(*=======================================================*)
	216:	(* Servobandeinzug rückwärts fahren, damit die Ausschiebezylinder das Band sicher erwischen *)
		IF fb_state_entry.E THEN
			axis_bandeinzug_achse.st_ctrl.in.b_ausfaedeln_servo := TRUE;
		END_IF

		(*-----------------------Weiterschaltbedingungen----------------------------*)
		IF axis_bandeinzug_achse.st_ctrl.out.b_ausgefaedelt_servo AND NOT fb_state_entry.E THEN
			axis_bandeinzug_achse.st_ctrl.in.b_ausfaedeln_servo := FALSE;
			fb_state_entry.i16_next_step := 217;(*Neu*)
		END_IF

(*=======================================================*)
	217:	(* Fänger ins Band fahren, damit die Bremse gelöst werden kann *)
		IF fb_state_entry.E THEN
				zyl_bawe_faenger_li.st_ctrl.in.b_ausfahren := TRUE;
		END_IF

		(*-----------------------Weiterschaltbedingungen----------------------------*)
		IF 	zyl_bawe_faenger_li.st_ctrl.out.b_ausgefahren AND
			gb_ba_auto_kontroller
			THEN
				zyl_bawe_faenger_li.st_ctrl.in.b_ausfahren := FALSE;
				fb_state_entry.i16_next_step := 218;
		END_IF

(*=======================================================*)
	218:	(* Bremse an Servobandeinzug lösen, damit Band heraus gezogen werden kann. Die Bestückachse hat die Slavekopplung bereits gelöst. *)
		IF fb_state_entry.E THEN
			axis_bandeinzug_achse.st_ctrl.in.b_bremse_auf := TRUE;
		END_IF

		(*-----------------------Weiterschaltbedingungen----------------------------*)
		IF axis_bandeinzug_achse.st_ctrl.out.b_bremse_geoeffnet AND NOT fb_state_entry.E THEN
			axis_bandeinzug_achse.st_ctrl.in.b_bremse_auf := FALSE;
			fb_state_entry.i16_next_step := 220;
		END_IF

(*=======================================================*)
	220:	(* Vorschub einfahren und Band aus WKZ rausziehen *)
		IF fb_state_entry.E THEN
			zyl_bawe_vorschub.st_ctrl.in.b_einfahren := TRUE;
			i16_akt_ausfaedeln := i16_akt_ausfaedeln + 1;
		END_IF

		(*-----------------------Weiterschaltbedingungen----------------------------*)
		IF zyl_bawe_vorschub.st_ctrl.out.b_eingefahren AND gb_ba_auto_kontroller THEN
			zyl_bawe_vorschub.st_ctrl.in.b_einfahren := FALSE;
			IF i16_akt_ausfaedeln <= i16_vorgabe_ausfaedeln THEN
				fb_state_entry.i16_next_step := 230;
			ELSE
				fb_state_entry.i16_next_step := 280;
			END_IF
		END_IF

(*=======================================================*)
	230:	(* Bandwechselhalter links ausfahren um Band nachfassen zu können *)
		IF fb_state_entry.E THEN
			zyl_bawe_halter_li.st_ctrl.in.b_ausfahren := TRUE;
		END_IF

		(*-----------------------Weiterschaltbedingungen----------------------------*)
		IF zyl_bawe_halter_li.st_ctrl.out.b_ausgefahren AND gb_ba_auto_kontroller THEN
			zyl_bawe_halter_li.st_ctrl.in.b_ausfahren := FALSE;
			fb_state_entry.i16_next_step := 240;
		END_IF

(*=======================================================*)
	240:	(* Bandwechselfänger links einfahren*)
		IF fb_state_entry.E THEN
			zyl_bawe_faenger_li.st_ctrl.in.b_einfahren := TRUE;
		END_IF

		(*-----------------------Weiterschaltbedingungen----------------------------*)
		IF zyl_bawe_faenger_li.st_ctrl.out.b_eingefahren AND gb_ba_auto_kontroller THEN
			zyl_bawe_faenger_li.st_ctrl.in.b_einfahren := FALSE;
			fb_state_entry.i16_next_step := 250;
		END_IF

(*=======================================================*)
	250:	(* Vorschub ausfahren und Band nachfassen *)
		IF fb_state_entry.E THEN
			zyl_bawe_vorschub.st_ctrl.in.b_ausfahren := TRUE;
		END_IF

		(*-----------------------Weiterschaltbedingungen----------------------------*)
		IF zyl_bawe_vorschub.st_ctrl.out.b_ausgefahren AND gb_ba_auto_kontroller THEN
			zyl_bawe_vorschub.st_ctrl.in.b_ausfahren := FALSE;
			fb_state_entry.i16_next_step := 260;
		END_IF

(*=======================================================*)
	260:	(* Bandwechselfänger links ausfahren zum Band halten *)
		IF fb_state_entry.E THEN
			zyl_bawe_faenger_li.st_ctrl.in.b_ausfahren := TRUE;
		END_IF

		(*-----------------------Weiterschaltbedingungen----------------------------*)
		IF zyl_bawe_faenger_li.st_ctrl.out.b_ausgefahren AND gb_ba_auto_kontroller THEN
			zyl_bawe_faenger_li.st_ctrl.in.b_ausfahren := FALSE;
			fb_state_entry.i16_next_step := 270;
		END_IF

(*=======================================================*)
	270:	(* Bandwechselhalter links einfahren und Band freigeben*)
		IF fb_state_entry.E THEN
			zyl_bawe_halter_li.st_ctrl.in.b_einfahren := TRUE;
		END_IF

		(*-----------------------Weiterschaltbedingungen----------------------------*)
		IF zyl_bawe_halter_li.st_ctrl.out.b_eingefahren AND gb_ba_auto_kontroller THEN
			zyl_bawe_halter_li.st_ctrl.in.b_einfahren := FALSE;
			fb_state_entry.i16_next_step := 220;
		END_IF

(*=======================================================*)
	280:	(* Fänger links einfahren zum Ausfädeln *)
		IF fb_state_entry.E THEN
			zyl_bawe_faenger_li.st_ctrl.in.b_einfahren := TRUE;
		END_IF

		(*-----------------------Weiterschaltbedingungen----------------------------*)
		IF zyl_bawe_faenger_li.st_ctrl.out.b_eingefahren AND gb_ba_auto_kontroller THEN
			zyl_bawe_faenger_li.st_ctrl.in.b_einfahren := FALSE;
			fb_state_entry.i16_next_step := 290;
		END_IF

(*=======================================================*)
	290:	(* Band ist herausgezogen - prüfe Einstellung bzw. Bandanwesenheit im rechten Einzug *)
		b_ausgefaedelt:=b_materialmangel;
			(* Band vorhanden -> Beginn automatischer Bandwechsel *)
		(*-----------------------Weiterschaltbedingungen----------------------------*)
		IF fb_tof_bandende_re.Q AND gst_datensatz.st_md.b_auto_Bandwechsel THEN
			b_spulenwechsel := TRUE;
			fb_state_entry.i16_next_step := 300;
		ELSE
			(* Bandherausziehen ist fertig *)
			fb_state_entry.i16_next_step := 295;
		END_IF

(*=======================================================*)
	291:	(* Bediener muss am Backpanel auswählen ob Bandwechsel oder Trennstelle *)

		(*-----------------------Weiterschaltbedingungen----------------------------*)
		IF visu_hinten.out.b_Bandwechsel THEN
			(* Band vorhanden -> Beginn automatischer Bandwechsel *)
			visu_hinten.in.b_bandwechsel_aktiv := FALSE;
			visu_hinten.in.current_visu_folie := 'BESTUECKZELLE_1700';
			fb_state_entry.i16_next_step := 300;
		ELSIF visu_hinten.out.b_Trennstelle THEN
			visu_hinten.in.b_bandwechsel_aktiv := FALSE;
			CASE gst_datensatz.st_wkz.i16_typ_bandeinzug OF

				 BANDWECHSLER_V2:
					visu_hinten.in.current_visu_folie := 'BA_1700_BAND_EINFAEDELN';

				SERVO:
					visu_hinten.in.current_visu_folie := 'BA1700_SERVO_BAND_EINFAEDELN';
			END_CASE
			fb_state_entry.i16_next_step := 295;
		END_IF

(*=======================================================*)
	295:	(* Vorschub ausfahren und fertig -> Band wird jetzt im gleichen Einzug manuell eingelegt mit Einfädelprozedur in der Bestückachse *)
		IF fb_state_entry.E THEN
			zyl_bawe_vorschub.st_ctrl.in.b_ausfahren := TRUE;
		END_IF

		(*-----------------------Weiterschaltbedingungen----------------------------*)
		IF zyl_bawe_vorschub.st_ctrl.out.b_ausgefahren AND gb_ba_auto_kontroller THEN
			zyl_bawe_vorschub.st_ctrl.in.b_ausfahren := FALSE;
			st_ctrl_out.b_fertig_2 := TRUE;
			fb_state_entry.i16_next_step := BEREIT;
		END_IF

(*=======================================================*)
	300:	(* Fänger rechts ausfahren *)
		IF fb_state_entry.E THEN
			zyl_bawe_faenger_re.st_ctrl.in.b_ausfahren := TRUE;
		END_IF

		(*-----------------------Weiterschaltbedingungen----------------------------*)
		IF 	zyl_bawe_faenger_re.st_ctrl.out.b_ausgefahren AND
			gb_ba_auto_kontroller
			THEN
				zyl_bawe_faenger_re.st_ctrl.in.b_ausfahren := FALSE;
				fb_state_entry.i16_next_step := 310;
		END_IF

(*=======================================================*)
	310:	(* Halter rechts einfahren *)
		IF fb_state_entry.E THEN
			zyl_bawe_halter_re.st_ctrl.in.b_einfahren := TRUE;
		END_IF

		(*-----------------------Weiterschaltbedingungen----------------------------*)
		IF zyl_bawe_halter_re.st_ctrl.out.b_eingefahren AND gb_ba_auto_kontroller THEN
			zyl_bawe_halter_re.st_ctrl.in.b_einfahren := FALSE;
			fb_state_entry.i16_next_step := 315;
		END_IF

(*=======================================================*)
	315:	(* Spulenbremse rechts oben? *)

		(*-----------------------Weiterschaltbedingungen----------------------------*)
		IF zyl_haspel_re_abspulen.st_ctrl.out.b_ausgefahren AND gb_ba_auto_kontroller THEN
			fb_state_entry.i16_next_step := 320;
		END_IF

(*=======================================================*)
	320:	(* Querschub ausfahren -> nach links und Haspeln nach links: Haspel verschieben ausfahren und Bandabzug einfahren *)
		IF fb_state_entry.E THEN
			zyl_bawe_querschub.st_ctrl.in.b_ausfahren := TRUE;
			zyl_haspel_verschieben.st_ctrl.in.b_ausfahren := TRUE;
			zyl_bandeinzuege_verschieben.st_ctrl.in.b_einfahren := TRUE;
		END_IF

		(*-----------------------Weiterschaltbedingungen----------------------------*)
		IF 	zyl_bawe_querschub.st_ctrl.out.b_ausgefahren AND
			zyl_haspel_verschieben.st_ctrl.out.b_ausgefahren AND
			zyl_bandeinzuege_verschieben.st_ctrl.out.b_eingefahren AND
			gb_ba_auto_kontroller
			THEN
				zyl_bawe_querschub.st_ctrl.in.b_ausfahren := FALSE;
				zyl_haspel_verschieben.st_ctrl.in.b_ausfahren := FALSE;
				zyl_bandeinzuege_verschieben.st_ctrl.in.b_einfahren := FALSE;
				CASE gst_datensatz.st_wkz.i16_typ_bandeinzug OF

					BANDWECHSLER_V2:
						fb_state_entry.i16_next_step := 330;

					SERVO:
						fb_state_entry.i16_next_step := 325;
				END_CASE
		END_IF

		IF fb_state_entry.X THEN
			b_spulenwechsel := FALSE;
		END_IF

(*=======================================================*)
	325:	(* Igelrad auf Position *)
		IF fb_state_entry.E THEN
			axis_bandeinzug_achse.st_ctrl.in.b_startpos := TRUE;
			fb_ton_wz.PT := t#100ms;
			fb_ton_wz.IN := TRUE;
		END_IF

		(*-----------------------Weiterschaltbedingungen----------------------------*)
		IF axis_bandeinzug_achse.st_ctrl.out.b_servo_auf_einfaedelpos
		AND gb_ba_auto_kontroller AND fb_ton_wz.Q THEN
			axis_bandeinzug_achse.st_ctrl.in.b_startpos := FALSE;
			fb_state_entry.i16_next_step := 330;
		END_IF

		IF fb_state_entry.X THEN
			fb_ton_wz.IN := FALSE;
		END_IF

(*=======================================================*)
	330:	(* Vorschub ausfahren *)
		IF fb_state_entry.E THEN
			zyl_bawe_vorschub.st_ctrl.in.b_ausfahren := TRUE;
			i16_akt_einfaedeln := i16_akt_einfaedeln + 1;
		END_IF

		(*-----------------------Weiterschaltbedingungen----------------------------*)
		IF zyl_bawe_vorschub.st_ctrl.out.b_ausgefahren AND gb_ba_auto_kontroller THEN
			zyl_bawe_vorschub.st_ctrl.in.b_ausfahren := FALSE;
			IF i16_akt_einfaedeln < i16_vorgabe_einfaedeln THEN
				fb_state_entry.i16_next_step := 340;
			ELSE
				fb_state_entry.i16_next_step := 390;		 (*mit Wartezeit alt 400*)
			END_IF
		END_IF

(*=======================================================*)
	340:	(* Halter rechts ausfahren *)
		IF fb_state_entry.E THEN
			zyl_bawe_halter_re.st_ctrl.in.b_ausfahren := TRUE;
		END_IF

		(*-----------------------Weiterschaltbedingungen----------------------------*)
		IF zyl_bawe_halter_re.st_ctrl.out.b_ausgefahren AND gb_ba_auto_kontroller THEN
			zyl_bawe_halter_re.st_ctrl.in.b_ausfahren := FALSE;
			fb_state_entry.i16_next_step := 350;
		END_IF

(*=======================================================*)
	350:	(* Fänger rechts einfahren *)
		IF fb_state_entry.E THEN
			zyl_bawe_faenger_re.st_ctrl.in.b_einfahren := TRUE;
		END_IF

		(*-----------------------Weiterschaltbedingungen----------------------------*)
		IF zyl_bawe_faenger_re.st_ctrl.out.b_eingefahren AND gb_ba_auto_kontroller THEN
			zyl_bawe_faenger_re.st_ctrl.in.b_einfahren := FALSE;
			fb_state_entry.i16_next_step := 360;
		END_IF

(*=======================================================*)
	360:	(* Vorschub einfahren *)
		IF fb_state_entry.E THEN
			zyl_bawe_vorschub.st_ctrl.in.b_einfahren := TRUE;
		END_IF

		(*-----------------------Weiterschaltbedingungen----------------------------*)
		IF zyl_bawe_vorschub.st_ctrl.out.b_eingefahren AND gb_ba_auto_kontroller THEN
			zyl_bawe_vorschub.st_ctrl.in.b_einfahren := FALSE;
			fb_state_entry.i16_next_step := 370;
		END_IF

(*=======================================================*)
	370:	(* Fänger rechts ausfahren *)
		IF fb_state_entry.E THEN
			zyl_bawe_faenger_re.st_ctrl.in.b_ausfahren := TRUE;
		END_IF

		(*-----------------------Weiterschaltbedingungen----------------------------*)
		IF zyl_bawe_faenger_re.st_ctrl.out.b_ausgefahren AND gb_ba_auto_kontroller THEN
			zyl_bawe_faenger_re.st_ctrl.in.b_ausfahren := FALSE;
			fb_state_entry.i16_next_step := 380;
		END_IF

(*=======================================================*)
	380:	(* Halter rechts einfahren *)
		IF fb_state_entry.E THEN
			zyl_bawe_halter_re.st_ctrl.in.b_einfahren := TRUE;
		END_IF

		(*-----------------------Weiterschaltbedingungen----------------------------*)
		IF zyl_bawe_halter_re.st_ctrl.out.b_eingefahren AND gb_ba_auto_kontroller THEN
			zyl_bawe_halter_re.st_ctrl.in.b_einfahren := FALSE;
			fb_state_entry.i16_next_step := 330;
		END_IF

(*=======================================================*)
	390:	(* Wartezeit damit der Fänger vom WZ trifft*)
		IF	 fb_state_entry.E THEN
			fb_ton_wz.IN:=FALSE;
		END_IF
		fb_ton_wz(IN:=TRUE,PT:=t#1000ms);
		(*-----------------------Weiterschaltbedingungen----------------------------*)
		IF 	fb_ton_wz.Q THEN
			fb_ton_wz.IN:=FALSE;
			fb_state_entry.i16_next_step := 400;
		END_IF

(*=======================================================*)
	400:	(* Nocken für Zylinder am Bandeinzug einschalten und somit Bandfänger ausfahren bzw. Bremse an Servobandeinzug wieder fest machen. *)

		CASE gst_datensatz.st_wkz.i16_typ_bandeinzug OF

			BANDWECHSLER_V2:

				IF fb_state_entry.E THEN
					(* Bandwechsler V2 ohne Sensoren und anderen Zylindern *)
					gst_datensatz.st_wkz.nockenschaltwerk_bestueckachse.arr_nocken[NO_BW_BANDFAENGER_BAWEV2_EINFAHREN].b_camvalid := TRUE;
					gst_datensatz.st_wkz.nockenschaltwerk_bestueckachse.arr_nocken[NO_BW_BANDFAENGER_BAWEV2_AUSFAHREN].b_camvalid := TRUE;
					gst_datensatz.st_wkz.nockenschaltwerk_bestueckachse.arr_nocken[NO_BW_BANDKLEMMEN_BAWEV2_EINFAHREN].b_camvalid := TRUE;
					gst_datensatz.st_wkz.nockenschaltwerk_bestueckachse.arr_nocken[NO_BW_BANDKLEMMEN_BAWEV2_AUSFAHREN].b_camvalid := TRUE;

					gst_datensatz.st_wkz.nockenschaltwerk_bestueckachse.arr_nocken[NO_PNEUMATIKBANDEINZUG_GLS].b_camvalid := TRUE;

					zyl_bandfaenger.fb.b_no_gesteuert_im_norm_betrieb := FALSE;
					zyl_bandklemmen.fb.b_no_gesteuert_im_norm_betrieb := FALSE;
					fb_ton_wz.PT := t#500ms;
					fb_ton_wz.IN := TRUE;
				END_IF

				(*-----------------------Weiterschaltbedingungen----------------------------*)
				IF fb_ton_wz.Q THEN
					fb_ton_wz.IN := FALSE;
					fb_state_entry.i16_next_step := 410;
				END_IF

			SERVO:
				IF fb_state_entry.E THEN
					axis_bandeinzug_achse.st_ctrl.in.b_bremse_auf := TRUE;	(* Bremse auf zum Position übernehmen *)
				END_IF

				(*-----------------------Weiterschaltbedingungen----------------------------*)
				IF axis_bandeinzug_achse.st_ctrl.out.b_bremse_geoeffnet THEN
					axis_bandeinzug_achse.st_ctrl.in.b_bremse_auf := FALSE;
					fb_state_entry.i16_next_step := 410;
				END_IF
		END_CASE;

(*=======================================================*)
	410:	(* Fänger rechts einfahren *)
		IF fb_state_entry.E THEN
			zyl_bawe_faenger_re.st_ctrl.in.b_einfahren := TRUE;
		END_IF

		(*-----------------------Weiterschaltbedingungen----------------------------*)
		IF zyl_bawe_faenger_re.st_ctrl.out.b_eingefahren
		AND gb_ba_auto_kontroller THEN
			zyl_bawe_faenger_re.st_ctrl.in.b_einfahren := FALSE;
			(* Bandwechsel ist fertig *)
			st_ctrl_out.b_fertig := TRUE;
			fb_state_entry.i16_next_step := BEREIT;
		END_IF


(*---------------------------------------------------------------------------------------------------------------------------------------------------------------------------------------------------*)
(*========================Bandeinzug rechts ist leer===============================*)
	500:	(* Fänger links ausfahren zum Band halten, Fänger rechts einfahren zur Bandfreigabe im rechten Einzug - Halter gegensinnig *)
		IF fb_state_entry.E THEN
			zyl_bawe_faenger_re.st_ctrl.in.b_ausfahren := TRUE;
			zyl_bawe_faenger_li.st_ctrl.in.b_einfahren := TRUE;
			zyl_bawe_halter_re.st_ctrl.in.b_einfahren := TRUE;
			zyl_bawe_halter_li.st_ctrl.in.b_ausfahren := TRUE;
		END_IF

		(*-----------------------Weiterschaltbedingungen----------------------------*)
		IF 	zyl_bawe_faenger_re.st_ctrl.out.b_ausgefahren AND
			zyl_bawe_faenger_li.st_ctrl.out.b_eingefahren AND
			zyl_bawe_halter_re.st_ctrl.out.b_eingefahren AND
			zyl_bawe_halter_li.st_ctrl.out.b_ausgefahren AND
			gb_ba_auto_kontroller
			THEN
				zyl_bawe_faenger_re.st_ctrl.in.b_ausfahren := FALSE;
				zyl_bawe_faenger_li.st_ctrl.in.b_einfahren := FALSE;
				zyl_bawe_halter_re.st_ctrl.in.b_einfahren := FALSE;
				zyl_bawe_halter_li.st_ctrl.in.b_ausfahren := FALSE;
				fb_state_entry.i16_next_step := 510;
		END_IF

(*=======================================================*)
	510:	(* Band-Zylinder einfahren bzw. Servobandeinzug lösen *)
		CASE gst_datensatz.st_wkz.i16_typ_bandeinzug OF
			BANDWECHSLER_V2:
				IF fb_state_entry.E THEN
					(* Zylinder einfahren *)
					zyl_bandfaenger.st_ctrl.in.b_einfahren := TRUE;
					zyl_bandklemmen.st_ctrl.in.b_einfahren := TRUE;
				END_IF

				(*-----------------------Weiterschaltbedingungen----------------------------*)
				IF 	zyl_bandfaenger.st_ctrl.out.b_eingefahren AND
					zyl_bandklemmen.st_ctrl.out.b_eingefahren AND
					gb_ba_auto_kontroller
					THEN
						zyl_bandfaenger.st_ctrl.in.b_einfahren := FALSE;
						zyl_bandklemmen.st_ctrl.in.b_einfahren := FALSE;
						fb_state_entry.i16_next_step := 520;
				END_IF

			SERVO:
				zyl_bawe_faenger_re.st_ctrl.in.b_einfahren := TRUE;
				zyl_bawe_halter_re.st_ctrl.in.b_einfahren := TRUE;
				(*-----------------------Weiterschaltbedingungen----------------------------*)
				IF 	zyl_bawe_faenger_re.st_ctrl.out.b_eingefahren AND
					zyl_bawe_halter_re.st_ctrl.out.b_eingefahren AND
					gb_ba_auto_kontroller
					THEN
						zyl_bawe_faenger_re.st_ctrl.in.b_einfahren := FALSE;
						zyl_bawe_halter_re.st_ctrl.in.b_einfahren := FALSE;
						fb_state_entry.i16_next_step := 516;
				END_IF
		END_CASE;

(*=======================================================*)
	516:	(* Servobandeinzug rückwärts fahren, damit die Ausschiebezylinder das Band sicher erwischen *)
		IF fb_state_entry.E THEN
			axis_bandeinzug_achse.st_ctrl.in.b_ausfaedeln_servo := TRUE;
		END_IF

		(*-----------------------Weiterschaltbedingungen----------------------------*)
		IF axis_bandeinzug_achse.st_ctrl.out.b_ausgefaedelt_servo AND NOT fb_state_entry.E THEN
			axis_bandeinzug_achse.st_ctrl.in.b_ausfaedeln_servo := FALSE;
			fb_state_entry.i16_next_step := 517;(*Neu*)
		END_IF

(*=======================================================*)
	517:	(* Fänger ins Band fahren, damit die Bremse gelöst werden kann *)
		IF fb_state_entry.E THEN
				zyl_bawe_faenger_re.st_ctrl.in.b_ausfahren := TRUE;
		END_IF

		(*-----------------------Weiterschaltbedingungen----------------------------*)
		IF 	zyl_bawe_faenger_re.st_ctrl.out.b_ausgefahren AND
			gb_ba_auto_kontroller
			THEN
				zyl_bawe_faenger_re.st_ctrl.in.b_ausfahren := FALSE;
				fb_state_entry.i16_next_step := 518;
		END_IF

(*=======================================================*)
	518:	(* Bremse an Servobandeinzug lösen, damit Band heraus gezogen werden kann. Die Bestückachse hat die Slavekopplung bereits gelöst. *)
		IF fb_state_entry.E THEN
			axis_bandeinzug_achse.st_ctrl.in.b_bremse_auf := TRUE;
		END_IF

		(*-----------------------Weiterschaltbedingungen----------------------------*)
		IF axis_bandeinzug_achse.st_ctrl.out.b_bremse_geoeffnet AND NOT fb_state_entry.E THEN
			axis_bandeinzug_achse.st_ctrl.in.b_bremse_auf := FALSE;
			fb_state_entry.i16_next_step := 520;
		END_IF

(*=======================================================*)
	520:	(* Vorschub einfahren und Band aus WKZ rausziehen *)
		IF fb_state_entry.E THEN
			zyl_bawe_vorschub.st_ctrl.in.b_einfahren := TRUE;
			i16_akt_ausfaedeln := i16_akt_ausfaedeln + 1;
		END_IF

		(*-----------------------Weiterschaltbedingungen----------------------------*)
		IF zyl_bawe_vorschub.st_ctrl.out.b_eingefahren AND gb_ba_auto_kontroller THEN
			zyl_bawe_vorschub.st_ctrl.in.b_einfahren := FALSE;
			IF i16_akt_ausfaedeln <= i16_vorgabe_ausfaedeln THEN
				fb_state_entry.i16_next_step := 530;
			ELSE
				fb_state_entry.i16_next_step := 580;
			END_IF
		END_IF

(*=======================================================*)
	530:	(* Bandwechselhalter rechts ausfahren um Band nachfassen zu können *)
		IF fb_state_entry.E THEN
			zyl_bawe_halter_re.st_ctrl.in.b_ausfahren := TRUE;
		END_IF

		(*-----------------------Weiterschaltbedingungen----------------------------*)
		IF zyl_bawe_halter_re.st_ctrl.out.b_ausgefahren AND gb_ba_auto_kontroller THEN
			zyl_bawe_halter_re.st_ctrl.in.b_ausfahren := FALSE;
			fb_state_entry.i16_next_step := 540;
		END_IF

(*=======================================================*)
	540:	(* Bandwechselfänger rechts einfahren*)
		IF fb_state_entry.E THEN
			zyl_bawe_faenger_re.st_ctrl.in.b_einfahren := TRUE;
		END_IF

		(*-----------------------Weiterschaltbedingungen----------------------------*)
		IF zyl_bawe_faenger_re.st_ctrl.out.b_eingefahren AND gb_ba_auto_kontroller THEN
			zyl_bawe_faenger_re.st_ctrl.in.b_einfahren := FALSE;
			fb_state_entry.i16_next_step := 550;
		END_IF

(*=======================================================*)
	550:	(* Vorschub ausfahren und Band nachfassen *)
		IF fb_state_entry.E THEN
			zyl_bawe_vorschub.st_ctrl.in.b_ausfahren := TRUE;
		END_IF

		(*-----------------------Weiterschaltbedingungen----------------------------*)
		IF zyl_bawe_vorschub.st_ctrl.out.b_ausgefahren AND gb_ba_auto_kontroller THEN
			zyl_bawe_vorschub.st_ctrl.in.b_ausfahren := FALSE;
			fb_state_entry.i16_next_step := 560;
		END_IF

(*=======================================================*)
	560:	(* Bandwechselfänger rechts ausfahren zum Band halten *)
		IF fb_state_entry.E THEN
			zyl_bawe_faenger_re.st_ctrl.in.b_ausfahren := TRUE;
		END_IF

		(*-----------------------Weiterschaltbedingungen----------------------------*)
		IF zyl_bawe_faenger_re.st_ctrl.out.b_ausgefahren AND gb_ba_auto_kontroller THEN
			zyl_bawe_faenger_re.st_ctrl.in.b_ausfahren := FALSE;
			fb_state_entry.i16_next_step := 570;
		END_IF

(*=======================================================*)
	570:	(* Bandwechselhalter rechts einfahren und Band freigeben*)
		IF fb_state_entry.E THEN
			zyl_bawe_halter_re.st_ctrl.in.b_einfahren := TRUE;
		END_IF

		(*-----------------------Weiterschaltbedingungen----------------------------*)
		IF zyl_bawe_halter_re.st_ctrl.out.b_eingefahren AND gb_ba_auto_kontroller THEN
			zyl_bawe_halter_re.st_ctrl.in.b_einfahren := FALSE;
			fb_state_entry.i16_next_step := 520;
		END_IF

(*=======================================================*)
	580:	(* Fänger rechts einfahren zum Ausfädeln *)
		IF fb_state_entry.E THEN
			zyl_bawe_faenger_re.st_ctrl.in.b_einfahren := TRUE;
		END_IF

		(*-----------------------Weiterschaltbedingungen----------------------------*)
		IF 	zyl_bawe_faenger_re.st_ctrl.out.b_eingefahren AND
			gb_ba_auto_kontroller
			THEN
				zyl_bawe_faenger_re.st_ctrl.in.b_einfahren := FALSE;
				fb_state_entry.i16_next_step := 590;
		END_IF

(*=======================================================*)
	590:	(* Band ist herausgezogen  - prüfe Einstellung bzw. Bandanwesenheit im linken Einzug *)
		b_ausgefaedelt:=b_materialmangel;
		(*-----------------------Weiterschaltbedingungen----------------------------*)
		IF fb_tof_bandende_li.Q  AND gst_datensatz.st_md.b_auto_Bandwechsel THEN
			b_spulenwechsel := TRUE;
			fb_state_entry.i16_next_step := 600;
		ELSE
			(* Bandherausziehen ist fertig *)
			fb_state_entry.i16_next_step := 595;
		END_IF

(*=======================================================*)
	591:	(* Bediener muss am Backpanel auswählen ob Bandwechsel oder Trennstelle *)

		(*-----------------------Weiterschaltbedingungen----------------------------*)
		IF visu_hinten.out.b_Bandwechsel THEN
			(* Band vorhanden -> Beginn automatischer Bandwechsel *)
			visu_hinten.in.b_bandwechsel_aktiv := FALSE;
			visu_hinten.in.current_visu_folie := 'BESTUECKZELLE_1700';
			fb_state_entry.i16_next_step := 600;
		ELSIF visu_hinten.out.b_Trennstelle THEN
			visu_hinten.in.b_bandwechsel_aktiv := FALSE;
			CASE gst_datensatz.st_wkz.i16_typ_bandeinzug OF

				BANDWECHSLER_V2:
					visu_hinten.in.current_visu_folie := 'BA_1700_BAND_EINFAEDELN';

				SERVO:
					visu_hinten.in.current_visu_folie := 'BA1700_SERVO_BAND_EINFAEDELN';
			END_CASE
			fb_state_entry.i16_next_step := 595;
		END_IF


(*=======================================================*)
	595:	(* Vorschub ausfahren und fertig -> Band wird jetzt im gleichen Einzug manuell eingelegt mit Einfädelprozedur in der Bestückachse *)
		IF fb_state_entry.E THEN
			zyl_bawe_vorschub.st_ctrl.in.b_ausfahren := TRUE;
		END_IF

		(*-----------------------Weiterschaltbedingungen----------------------------*)
		IF zyl_bawe_vorschub.st_ctrl.out.b_ausgefahren AND gb_ba_auto_kontroller THEN
			zyl_bawe_vorschub.st_ctrl.in.b_ausfahren := FALSE;
			st_ctrl_out.b_fertig_2 := TRUE;
			fb_state_entry.i16_next_step := BEREIT;
		END_IF

(*=======================================================*)
	600:	(* Fänger links ausfahren *)
		IF fb_state_entry.E THEN
			zyl_bawe_faenger_li.st_ctrl.in.b_ausfahren := TRUE;
		END_IF

		(*-----------------------Weiterschaltbedingungen----------------------------*)
		IF 	zyl_bawe_faenger_li.st_ctrl.out.b_ausgefahren AND
			gb_ba_auto_kontroller
			THEN
				zyl_bawe_faenger_li.st_ctrl.in.b_ausfahren := FALSE;
				fb_state_entry.i16_next_step := 610;
		END_IF

(*=======================================================*)
	610:	(* Halter links einfahren *)
		IF fb_state_entry.E THEN
			zyl_bawe_halter_li.st_ctrl.in.b_einfahren := TRUE;
		END_IF

		(*-----------------------Weiterschaltbedingungen----------------------------*)
		IF zyl_bawe_halter_li.st_ctrl.out.b_eingefahren AND gb_ba_auto_kontroller THEN
			zyl_bawe_halter_li.st_ctrl.in.b_einfahren := FALSE;
			fb_state_entry.i16_next_step := 615;
		END_IF

(*=======================================================*)
	615:	(* Spulenbremse links oben? *)

		(*-----------------------Weiterschaltbedingungen----------------------------*)
		IF zyl_haspel_li_abspulen.st_ctrl.out.b_ausgefahren AND gb_ba_auto_kontroller THEN
			fb_state_entry.i16_next_step := 620;
		END_IF

(*=======================================================*)
	620:	(* Querschub einfahren -> nach rechts und Haspeln nach rechts: Haspel verschieben einfahren und Bandabzug ausfahren*)
		IF fb_state_entry.E THEN
			zyl_bawe_querschub.st_ctrl.in.b_einfahren := TRUE;
			zyl_haspel_verschieben.st_ctrl.in.b_einfahren := TRUE;
			zyl_bandeinzuege_verschieben.st_ctrl.in.b_ausfahren := TRUE;
		END_IF

		(*-----------------------Weiterschaltbedingungen----------------------------*)
		IF 	zyl_bawe_querschub.st_ctrl.out.b_eingefahren AND
			zyl_haspel_verschieben.st_ctrl.out.b_eingefahren AND
			zyl_bandeinzuege_verschieben.st_ctrl.out.b_ausgefahren AND
			gb_ba_auto_kontroller
			THEN
				zyl_bawe_querschub.st_ctrl.in.b_einfahren := FALSE;
				zyl_haspel_verschieben.st_ctrl.in.b_einfahren := FALSE;
				zyl_bandeinzuege_verschieben.st_ctrl.in.b_ausfahren := FALSE;
				CASE gst_datensatz.st_wkz.i16_typ_bandeinzug OF

					BANDWECHSLER_V2:
						fb_state_entry.i16_next_step := 630;

					SERVO:
						fb_state_entry.i16_next_step := 625;
				END_CASE
		END_IF

		IF fb_state_entry.X THEN
			b_spulenwechsel := FALSE;
		END_IF

(*=======================================================*)
	625:	(* Igelrad auf Position *)
		IF fb_state_entry.E THEN
			axis_bandeinzug_achse.st_ctrl.in.b_startpos := TRUE;
			fb_ton_wz.PT := t#100ms;
			fb_ton_wz.IN := TRUE;
		END_IF

		(*-----------------------Weiterschaltbedingungen----------------------------*)
		IF axis_bandeinzug_achse.st_ctrl.out.b_servo_auf_einfaedelpos
			AND gb_ba_auto_kontroller AND fb_ton_wz.Q THEN
			axis_bandeinzug_achse.st_ctrl.in.b_startpos := FALSE;
			fb_state_entry.i16_next_step := 630;
		END_IF

		IF fb_state_entry.X THEN
			fb_ton_wz.IN := FALSE;
		END_IF

(*=======================================================*)
	630:	(* Vorschub ausfahren *)
		IF fb_state_entry.E THEN
			zyl_bawe_vorschub.st_ctrl.in.b_ausfahren := TRUE;
			i16_akt_einfaedeln := i16_akt_einfaedeln + 1;
		END_IF

		(*-----------------------Weiterschaltbedingungen----------------------------*)
		IF zyl_bawe_vorschub.st_ctrl.out.b_ausgefahren AND gb_ba_auto_kontroller THEN
			zyl_bawe_vorschub.st_ctrl.in.b_ausfahren := FALSE;
			IF i16_akt_einfaedeln < i16_vorgabe_einfaedeln THEN
				fb_state_entry.i16_next_step := 640;
			ELSE
				fb_state_entry.i16_next_step := 690; (*mit Wartezeit alt auf 700*)
			END_IF
		END_IF

(*=======================================================*)
	640:	(* Halter links ausfahren *)
		IF fb_state_entry.E THEN
			zyl_bawe_halter_li.st_ctrl.in.b_ausfahren := TRUE;
		END_IF

		(*-----------------------Weiterschaltbedingungen----------------------------*)
		IF zyl_bawe_halter_li.st_ctrl.out.b_ausgefahren AND gb_ba_auto_kontroller THEN
			zyl_bawe_halter_li.st_ctrl.in.b_ausfahren := FALSE;
			fb_state_entry.i16_next_step := 650;
		END_IF

(*=======================================================*)
	650:	(* Fänger links einfahren *)
		IF fb_state_entry.E THEN
			zyl_bawe_faenger_li.st_ctrl.in.b_einfahren := TRUE;
		END_IF

		(*-----------------------Weiterschaltbedingungen----------------------------*)
		IF zyl_bawe_faenger_li.st_ctrl.out.b_eingefahren AND gb_ba_auto_kontroller THEN
			zyl_bawe_faenger_li.st_ctrl.in.b_einfahren := FALSE;
			fb_state_entry.i16_next_step := 660;
		END_IF

(*=======================================================*)
	660:	(* Vorschub einfahren *)
		IF fb_state_entry.E THEN
			zyl_bawe_vorschub.st_ctrl.in.b_einfahren := TRUE;
		END_IF

		(*-----------------------Weiterschaltbedingungen----------------------------*)
		IF zyl_bawe_vorschub.st_ctrl.out.b_eingefahren AND gb_ba_auto_kontroller THEN
			zyl_bawe_vorschub.st_ctrl.in.b_einfahren := FALSE;
			fb_state_entry.i16_next_step := 670;
		END_IF

(*=======================================================*)
	670:	(* Fänger links ausfahren *)
		IF fb_state_entry.E THEN
			zyl_bawe_faenger_li.st_ctrl.in.b_ausfahren := TRUE;
		END_IF

		(*-----------------------Weiterschaltbedingungen----------------------------*)
		IF zyl_bawe_faenger_li.st_ctrl.out.b_ausgefahren AND gb_ba_auto_kontroller THEN
			zyl_bawe_faenger_li.st_ctrl.in.b_ausfahren := FALSE;
			fb_state_entry.i16_next_step := 680;
		END_IF

(*=======================================================*)
	680:	(* Halter links einfahren *)
		IF fb_state_entry.E THEN
			zyl_bawe_halter_li.st_ctrl.in.b_einfahren := TRUE;
		END_IF

		(*-----------------------Weiterschaltbedingungen----------------------------*)
		IF zyl_bawe_halter_li.st_ctrl.out.b_eingefahren AND gb_ba_auto_kontroller THEN
			zyl_bawe_halter_li.st_ctrl.in.b_einfahren := FALSE;
			fb_state_entry.i16_next_step := 630;
		END_IF
(*=======================================================*)
	690:	(* Wartezeit damit der Fänger vom WZ trifft*)
		IF	 fb_state_entry.E THEN
			fb_ton_wz.IN:=FALSE;
		END_IF
		fb_ton_wz(IN:=TRUE,PT:=t#1000ms);
		(*-----------------------Weiterschaltbedingungen----------------------------*)
		IF 	fb_ton_wz.Q THEN
			fb_ton_wz.IN:=FALSE;
			fb_state_entry.i16_next_step := 700;
		END_IF

(*=======================================================*)
	700:	(* Nocken für Zylinder am Bandeinzug einschalten und somit Bandfänger ausfahren bzw. Bremse an Servobandeinzug wieder fest machen. *)
		CASE gst_datensatz.st_wkz.i16_typ_bandeinzug OF

			BANDWECHSLER_V2:

				IF fb_state_entry.E THEN
					(* Bandwechsler V2 ohne Sensoren und anderen Zylindern *)
					gst_datensatz.st_wkz.nockenschaltwerk_bestueckachse.arr_nocken[NO_BW_BANDFAENGER_BAWEV2_EINFAHREN].b_camvalid := TRUE;
					gst_datensatz.st_wkz.nockenschaltwerk_bestueckachse.arr_nocken[NO_BW_BANDFAENGER_BAWEV2_AUSFAHREN].b_camvalid := TRUE;
					gst_datensatz.st_wkz.nockenschaltwerk_bestueckachse.arr_nocken[NO_BW_BANDKLEMMEN_BAWEV2_EINFAHREN].b_camvalid := TRUE;
					gst_datensatz.st_wkz.nockenschaltwerk_bestueckachse.arr_nocken[NO_BW_BANDKLEMMEN_BAWEV2_AUSFAHREN].b_camvalid := TRUE;

					gst_datensatz.st_wkz.nockenschaltwerk_bestueckachse.arr_nocken[NO_PNEUMATIKBANDEINZUG_GLS].b_camvalid := TRUE;

					zyl_bandfaenger.fb.b_no_gesteuert_im_norm_betrieb := FALSE;
					zyl_bandklemmen.fb.b_no_gesteuert_im_norm_betrieb := FALSE;
					fb_ton_wz.PT := t#500ms;
					fb_ton_wz.IN := TRUE;
				END_IF
		
				(*-----------------------Weiterschaltbedingungen----------------------------*)
				IF fb_ton_wz.Q THEN
					fb_ton_wz.IN := FALSE;
					fb_state_entry.i16_next_step := 710;
				END_IF

			SERVO:
				IF fb_state_entry.E THEN
					axis_bandeinzug_achse.st_ctrl.in.b_bremse_auf := TRUE;	(* Bremse auf zum Position übernehmen *)
				END_IF

				(*-----------------------Weiterschaltbedingungen----------------------------*)
				IF axis_bandeinzug_achse.st_ctrl.out.b_bremse_geoeffnet THEN
					axis_bandeinzug_achse.st_ctrl.in.b_bremse_auf := FALSE;
					fb_state_entry.i16_next_step := 710;
				END_IF
		END_CASE;

(*=======================================================*)
	710:	(* Fänger links einfahren *)
		IF fb_state_entry.E THEN
			zyl_bawe_faenger_li.st_ctrl.in.b_einfahren := TRUE;
		END_IF

		(*-----------------------Weiterschaltbedingungen----------------------------*)
		IF zyl_bawe_faenger_li.st_ctrl.out.b_eingefahren
		AND gb_ba_auto_kontroller THEN
			zyl_bawe_faenger_li.st_ctrl.in.b_einfahren := FALSE;
			(* Bandwechsel ist fertig *)
			st_ctrl_out.b_fertig := TRUE;
			fb_state_entry.i16_next_step := BEREIT;
		END_IF

(*=======================================================*)
	FEHLER:
		IF fb_state_entry.E THEN
			st_ctrl_out.b_fehler := TRUE;
			fb_ton_quitt.IN := FALSE;
			zyl_bawe_vorschub.st_ctrl.in.b_quittieren := FALSE;
			zyl_bawe_querschub.st_ctrl.in.b_quittieren := FALSE;
			zyl_bawe_faenger_li.st_ctrl.in.b_quittieren := FALSE;
			zyl_bawe_faenger_re.st_ctrl.in.b_quittieren := FALSE;
			zyl_bawe_halter_li.st_ctrl.in.b_quittieren := FALSE;
			zyl_bawe_halter_re.st_ctrl.in.b_quittieren := FALSE;
			zyl_haspel_verschieben.st_ctrl.in.b_quittieren := FALSE;
			zyl_bandeinzuege_verschieben.st_ctrl.in.b_quittieren := FALSE;
		END_IF

		(*-----------------------Weiterschaltbedingungen----------------------------*)
		IF st_ctrl_in.b_quitt AND NOT fb_state_entry.E THEN
			st_ctrl_out.b_fehler := TRUE;
			zyl_bawe_vorschub.st_ctrl.in.b_quittieren := TRUE;
			zyl_bawe_querschub.st_ctrl.in.b_quittieren := TRUE;
			zyl_bawe_faenger_li.st_ctrl.in.b_quittieren := TRUE;
			zyl_bawe_faenger_re.st_ctrl.in.b_quittieren := TRUE;
			zyl_bawe_halter_li.st_ctrl.in.b_quittieren := TRUE;
			zyl_bawe_halter_re.st_ctrl.in.b_quittieren := TRUE;
			zyl_haspel_verschieben.st_ctrl.in.b_quittieren := TRUE;
			zyl_bandeinzuege_verschieben.st_ctrl.in.b_quittieren := TRUE;
			fb_ton_quitt.IN := TRUE;
		END_IF

		IF fb_ton_quitt.Q THEN
			fb_ton_quitt.IN := FALSE;
			fb_state_entry.i16_next_step := INIT;
		END_IF

(*=======================================================*)
	STOP:
		IF fb_state_entry.E THEN
			fb_ton_quitt.IN := FALSE;
			zyl_bawe_vorschub.st_ctrl.in.b_quittieren := FALSE;
			zyl_bawe_querschub.st_ctrl.in.b_quittieren := FALSE;
			zyl_bawe_faenger_li.st_ctrl.in.b_quittieren := FALSE;
			zyl_bawe_faenger_re.st_ctrl.in.b_quittieren := FALSE;
			zyl_bawe_halter_li.st_ctrl.in.b_quittieren := FALSE;
			zyl_bawe_halter_re.st_ctrl.in.b_quittieren := FALSE;
			zyl_haspel_verschieben.st_ctrl.in.b_quittieren := FALSE;
			zyl_bandeinzuege_verschieben.st_ctrl.in.b_quittieren := FALSE;
		END_IF

		(*-----------------------Weiterschaltbedingungen----------------------------*)
		IF st_ctrl_in.b_quitt AND NOT fb_state_entry.E THEN
			fb_ton_quitt.IN := TRUE;
			zyl_bawe_vorschub.st_ctrl.in.b_quittieren := TRUE;
			zyl_bawe_querschub.st_ctrl.in.b_quittieren := TRUE;
			zyl_bawe_faenger_li.st_ctrl.in.b_quittieren := TRUE;
			zyl_bawe_faenger_re.st_ctrl.in.b_quittieren := TRUE;
			zyl_bawe_halter_li.st_ctrl.in.b_quittieren := TRUE;
			zyl_bawe_halter_re.st_ctrl.in.b_quittieren := TRUE;
			zyl_haspel_verschieben.st_ctrl.in.b_quittieren := TRUE;
			zyl_bandeinzuege_verschieben.st_ctrl.in.b_quittieren := TRUE;
		END_IF

		IF fb_ton_quitt.Q THEN
			fb_ton_quitt.IN := FALSE;
			fb_state_entry.i16_next_step := INIT;
		END_IF
END_CASE

fb_state_entry(
	i16_next_step:= , 
	i16_pos:= 2,
	s_debugtext:= ,
	E=> ,
	X=> , 
	i16_step=> ,
	i16_last_step=> );

IF st_config.b_config_fertig THEN
	(* Fehlermeldungen und Betriebsmeldungen ab dem Startindex in die globalen Meldungsarrays schreiben *)
	garr_stoermeldungen[st_config.i16_meld_startindex + 0] := sm_halter_nicht_oben;
	garr_stoermeldungen[st_config.i16_meld_startindex + 1] := sm_bandwechsel_ohne_ende;
	garr_stoermeldungen[st_config.i16_meld_startindex + 2] := sm_kein_band_anderer_einzug;
	garr_stoermeldungen[st_config.i16_meld_startindex + 3] := sm_kein_band_in_akt_einzug;
	garr_stoermeldungen[st_config.i16_meld_startindex + 4] := FALSE;
	garr_stoermeldungen[st_config.i16_meld_startindex + 5] := FALSE;
	garr_stoermeldungen[st_config.i16_meld_startindex + 6] := FALSE;
	garr_stoermeldungen[st_config.i16_meld_startindex + 7] := FALSE;
	garr_stoermeldungen[st_config.i16_meld_startindex + 8] := FALSE;
	garr_stoermeldungen[st_config.i16_meld_startindex + 9] := FALSE;
	garr_stoermeldungen[st_config.i16_meld_startindex + 10] := FALSE;
	garr_stoermeldungen[st_config.i16_meld_startindex + 11] := FALSE;
	garr_stoermeldungen[st_config.i16_meld_startindex + 12] := FALSE;
	garr_stoermeldungen[st_config.i16_meld_startindex + 13] := FALSE;
	garr_stoermeldungen[st_config.i16_meld_startindex + 14] := FALSE;
	garr_stoermeldungen[st_config.i16_meld_startindex + 15] := FALSE;
	garr_stoermeldungen[st_config.i16_meld_startindex + 16] := FALSE;
	garr_stoermeldungen[st_config.i16_meld_startindex + 17] := FALSE;
	garr_stoermeldungen[st_config.i16_meld_startindex + 18] := FALSE;
	garr_stoermeldungen[st_config.i16_meld_startindex + 19] := FALSE;
	
	garr_betriebsmeldungen[st_config.i16_meld_startindex + 0] := bm_bandwechselvorgang;
	garr_betriebsmeldungen[st_config.i16_meld_startindex + 1] := bm_bandwechsel_manuell;
	garr_betriebsmeldungen[st_config.i16_meld_startindex + 2] := FALSE;
	garr_betriebsmeldungen[st_config.i16_meld_startindex + 3] := FALSE;
	garr_betriebsmeldungen[st_config.i16_meld_startindex + 4] := FALSE;
	garr_betriebsmeldungen[st_config.i16_meld_startindex + 5] := FALSE;
	garr_betriebsmeldungen[st_config.i16_meld_startindex + 6] := FALSE;
	garr_betriebsmeldungen[st_config.i16_meld_startindex + 7] := FALSE;
	garr_betriebsmeldungen[st_config.i16_meld_startindex + 8] := FALSE;
	garr_betriebsmeldungen[st_config.i16_meld_startindex + 9] := FALSE;
	garr_betriebsmeldungen[st_config.i16_meld_startindex + 10] := FALSE;
	garr_betriebsmeldungen[st_config.i16_meld_startindex + 11] := FALSE;
	garr_betriebsmeldungen[st_config.i16_meld_startindex + 12] := FALSE;
	garr_betriebsmeldungen[st_config.i16_meld_startindex + 13] := FALSE;
	garr_betriebsmeldungen[st_config.i16_meld_startindex + 14] := FALSE;
	garr_betriebsmeldungen[st_config.i16_meld_startindex + 15] := FALSE;
	garr_betriebsmeldungen[st_config.i16_meld_startindex + 16] := FALSE;
	garr_betriebsmeldungen[st_config.i16_meld_startindex + 17] := FALSE;
	garr_betriebsmeldungen[st_config.i16_meld_startindex + 18] := FALSE;
	garr_betriebsmeldungen[st_config.i16_meld_startindex + 19] := FALSE;
END_IF
END_PROGRAM

(* POU Gemeinsamkeiten17xx/Werkzeug/ST_WkzAbsicherung, ST *)
PROGRAM ST_WkzAbsicherung
VAR_INPUT
	st_config								: struct_config;
	st_ctrl_in								: struct_ctrl_in;
END_VAR
VAR_IN_OUT
	st_visu								: struct_visu;
END_VAR
VAR_OUTPUT
	st_ctrl_out							: struct_ctrl_out;
END_VAR
VAR
	fb_ton_wz							: TON;
	fb_ton_uez							: TON;
	fb_ton_quitt							: TON;
	fb_state_entry							: ST_StateEntry;
	b_signalmerker_bestueckschieber_on		: BOOL := FALSE;
	b_signalmerker_bestueckschieber_off		: BOOL := FALSE;
	fb_r_trig_signal_bestueckschieber		: R_TRIG;
	fb_f_trig_signal_bestueckschieber		: F_TRIG;
	fb_r_trig_nocke_uw_bestueckschieber	: R_TRIG;
	fb_f_trig_nocke_uw_bestueckschieber	: F_TRIG;

	(* Eingänge *)
	(* BSV 1720 6-fach *)
	e_wkz_sicherung_niederhalter_li			AT %I* : BOOL;
	e_wkz_sicherung_faenger_li			AT %I* : BOOL;
	e_wkz_sicherung_abfallpodest_li		AT %I* : BOOL;
	e_wkz_sicherung_niederhalter_re		AT %I* : BOOL;
	e_wkz_sicherung_faenger_re			AT %I* : BOOL;
	e_wkz_sicherung_abfallpodest_re		AT %I* : BOOL;
	(* Erkennung/Kodierung für alte WKZ z.B. 1708alt *)
	e_kodierung_alt_wkz					AT %I* : BOOL;
	(* BSH 1700 *)
	e_wkz_sicherung_faenger				AT %I* : BOOL;
	e_bestueckschieber_ueberwachung		AT %I* : BOOL;

	(* Meldungen *)
	(* BSV 1720 6-fach *)
	sm_wkz_sicherung_niederhalter_li		: BOOL := FALSE;
	sm_wkz_sicherung_faenger_li			: BOOL := FALSE;
	sm_wkz_sicherung_abfallpodest_li		: BOOL := FALSE;
	sm_wkz_sicherung_niederhalter_re		: BOOL := FALSE;
	sm_wkz_sicherung_faenger_re			: BOOL := FALSE;
	sm_wkz_sicherung_abfallpodest_re		: BOOL := FALSE;
	(* BSH 1700 *)
	sm_wkz_sicherung_faenger				: BOOL := FALSE;
	sm_bestueckschieber_ueberwachung	: BOOL := FALSE;
	UW_Bestueckschieber_on: BOOL;
END_VAR
(* Zeiten *)
fb_ton_wz(IN:= , PT:= , Q=>  , ET=> );
fb_ton_uez(IN:= , PT:= , Q=>  , ET=> );
fb_ton_quitt(IN:= , PT:= t#100ms, Q=> , ET=> );

(* Flanken *)

fb_f_trig_nocke_uw_bestueckschieber(CLK:= nockenschaltwerk_bestueckachse.fb.arr_spur[SP_UW_BESTUECKSCHIEBER_ON], Q=> );
fb_r_trig_nocke_uw_bestueckschieber(CLK:= nockenschaltwerk_bestueckachse.fb.arr_spur[SP_UW_BESTUECKSCHIEBER_ON], Q=> );
fb_r_trig_signal_bestueckschieber(CLK:= e_bestueckschieber_ueberwachung, Q=> );
fb_f_trig_signal_bestueckschieber(CLK:= e_bestueckschieber_ueberwachung, Q=> );

UW_Bestueckschieber_on:=nockenschaltwerk_bestueckachse.fb.arr_spur[SP_UW_BESTUECKSCHIEBER_ON]; 	(*für Trace*)
(* Toplevel *)
IF fb_state_entry.i16_next_step > INIT AND fb_state_entry.i16_next_step < FEHLER THEN
	IF fb_state_entry.i16_next_step < STOP THEN
		IF st_ctrl_in.b_stop THEN
			fb_state_entry.i16_next_step := STOP;
		END_IF
	END_IF
END_IF

(* ======================================Schrittkette======================================== *)
fb_state_entry(
	i16_next_step:= ,
	i16_pos:= 1,
	s_debugtext:= ,
	E=> ,
	X=> ,
	i16_step=> ,
	i16_last_step=> );

CASE fb_state_entry.i16_step OF
(*=======================================================*)
	INIT_OBJ:
		IF st_config.b_config_fertig THEN
			fb_state_entry.i16_next_step := INIT;
		END_IF

(*=======================================================*)
	INIT:
		IF fb_state_entry.E THEN
			fb_ton_wz.IN := FALSE;
			fb_ton_uez.IN	:= FALSE;
			fb_ton_quitt.IN	 := FALSE;
			b_signalmerker_bestueckschieber_on := FALSE;
			b_signalmerker_bestueckschieber_off := FALSE;
			sm_wkz_sicherung_niederhalter_li := FALSE;
			sm_wkz_sicherung_faenger_li := FALSE;
			sm_wkz_sicherung_abfallpodest_li := FALSE;
			sm_wkz_sicherung_niederhalter_re := FALSE;
			sm_wkz_sicherung_faenger_re := FALSE;
			sm_wkz_sicherung_abfallpodest_re := FALSE;
			sm_wkz_sicherung_faenger := FALSE;
			sm_bestueckschieber_ueberwachung := FALSE;
			st_ctrl_out.b_fehler := FALSE;
			st_ctrl_out.b_bereit := FALSE;
			st_ctrl_out.b_fertig := FALSE;
			st_ctrl_out.b_einzelfertigung := FALSE;
		END_IF

		(*-----------------------Weiterschaltbedingungen----------------------------*)
		IF st_ctrl_in.b_init THEN
			fb_state_entry.i16_next_step := BEREIT;
		END_IF

(*=======================================================*)
	BEREIT:
		IF fb_state_entry.E THEN
			st_ctrl_out.b_bereit := TRUE;
		END_IF

		CASE gst_datensatz.st_md.i16_typ_zelle OF
			KEINE_ZELLE:
				;

			BESTUECKZELLE_1700:
				IF NOT gst_datensatz.st_md.b_wt_transport_simulation THEN
					IF NOT e_wkz_sicherung_faenger THEN
						sm_wkz_sicherung_faenger := TRUE;
						fb_state_entry.i16_next_step := FEHLER;
					END_IF

					IF ST_Virtuelle_Masterachse.fb_state_entry.i16_step >= BEREIT THEN
						IF gst_datensatz.st_bestueckprogramm.i16_b[ST_Virtuelle_Masterachse.i16_bestueckposzaehler] <> 0 THEN	(* Bei Umfahrung = 0 bewegt sich der Bestückschieber nicht *)
							(* Nocken werden in virtueller Bestückachse nach ein paar Hüben ausgeschaltet *)
							IF	(nockenschaltwerk_bestueckachse.fb.arr_spur[SP_UW_BESTUECKSCHIEBER_ON] AND  NOT e_bestueckschieber_ueberwachung) OR
								(nockenschaltwerk_bestueckachse.fb.arr_spur[SP_UW_BESTUECKSCHIEBER_OFF] AND e_bestueckschieber_ueberwachung)
								THEN
									sm_bestueckschieber_ueberwachung := TRUE;
									fb_state_entry.i16_next_step := FEHLER;
							END_IF
						END_IF
					END_IF


					(* Option: Flankenauswertung der GLS am Bestückschieber *)
(*					IF	nockenschaltwerk_bestueckachse.fb.arr_spur[SP_UW_BESTUECKSCHIEBER_ON] THEN
						IF 	fb_r_trig_signal_bestueckschieber.Q THEN
							b_signalmerker_bestueckschieber_on := TRUE;
						END_IF
						IF	 fb_f_trig_signal_bestueckschieber.Q THEN
							b_signalmerker_bestueckschieber_off := TRUE;
						END_IF
					END_IF

					(* Option: Beide setzen wenn Nocke abgeschaltet ist *)
					IF	NOT gst_datensatz.st_wkz.nockenschaltwerk_bestueckachse.arr_nocken[SP_UW_BESTUECKSCHIEBER_OFF].b_camvalid THEN
						b_signalmerker_bestueckschieber_on := TRUE;
						b_signalmerker_bestueckschieber_off := TRUE;
					END_IF

					IF 	fb_f_trig_nocke_uw_bestueckschieber.Q THEN

						IF 	b_signalmerker_bestueckschieber_off  AND
							b_signalmerker_bestueckschieber_on THEN
							b_signalmerker_bestueckschieber_on := FALSE;
							b_signalmerker_bestueckschieber_off := FALSE;
						ELSE
							sm_bestueckschieber_ueberwachung := TRUE;
							fb_state_entry.i16_next_step := FEHLER;
						END_IF
					END_IF
*)
				END_IF

			BESTUECKZELLE_1720:
				IF NOT gst_datensatz.st_md.b_wt_transport_simulation THEN
					IF e_kodierung_alt_wkz THEN
						(* BSV 1720 2-fach *)
						IF NOT  e_wkz_sicherung_faenger_li THEN
							sm_wkz_sicherung_faenger_li := TRUE;
							fb_state_entry.i16_next_step := FEHLER;
						END_IF
						IF NOT  e_wkz_sicherung_faenger_re THEN
							sm_wkz_sicherung_faenger_re := TRUE;
							fb_state_entry.i16_next_step := FEHLER;
						END_IF
					ELSE
						(* BSV 1720 6-fach *)
						IF	NOT ST_TippTasten.b_einfaedeln_aktiv THEN
							IF e_wkz_sicherung_niederhalter_li AND nockenschaltwerk_bestueckachse.fb.arr_spur[SP_UW_WKZ_NIEDERHALTER_LI] THEN
								sm_wkz_sicherung_niederhalter_li := TRUE;
								fb_state_entry.i16_next_step := 200;
							END_IF
							IF e_wkz_sicherung_niederhalter_re AND nockenschaltwerk_bestueckachse.fb.arr_spur[SP_UW_WKZ_NIEDERHALTER_RE] THEN
								sm_wkz_sicherung_niederhalter_re := TRUE;
								fb_state_entry.i16_next_step := 200;
							END_IF
						END_IF
						IF NOT  e_wkz_sicherung_faenger_li THEN
							sm_wkz_sicherung_faenger_li := TRUE;
							fb_state_entry.i16_next_step := FEHLER;
						END_IF
						IF NOT  e_wkz_sicherung_faenger_re THEN
							sm_wkz_sicherung_faenger_re := TRUE;
							fb_state_entry.i16_next_step := FEHLER;
						END_IF
						IF NOT e_wkz_sicherung_abfallpodest_li THEN
							sm_wkz_sicherung_abfallpodest_li := TRUE;
							fb_state_entry.i16_next_step := 200;
						END_IF
						IF NOT e_wkz_sicherung_abfallpodest_re THEN
							sm_wkz_sicherung_abfallpodest_re := TRUE;
							fb_state_entry.i16_next_step := 200;
						END_IF
					END_IF
				END_IF

			RASTERFOLIE:
				;
		END_CASE

(*=======================================================*)
	200:	(* Nur aktiv bei 1720 und WKZ-Absicherung 6-fach. Verzweigen nach Fehler erst, wenn OT erreicht wird - leichtere Fehlerbehebung. *)

		IF NOT gst_datensatz.st_md.b_wt_transport_simulation THEN
			(* BSV 1720 6-fach *)
			IF e_wkz_sicherung_niederhalter_li AND nockenschaltwerk_bestueckachse.fb.arr_spur[SP_UW_WKZ_NIEDERHALTER_LI] THEN
				sm_wkz_sicherung_niederhalter_li := TRUE;
			END_IF
			IF NOT  e_wkz_sicherung_faenger_li THEN
				sm_wkz_sicherung_faenger_li := TRUE;
				fb_state_entry.i16_next_step := FEHLER;
			END_IF
			IF NOT e_wkz_sicherung_abfallpodest_li THEN
				sm_wkz_sicherung_abfallpodest_li := TRUE;
			END_IF
			IF e_wkz_sicherung_niederhalter_re AND nockenschaltwerk_bestueckachse.fb.arr_spur[SP_UW_WKZ_NIEDERHALTER_RE] THEN
				sm_wkz_sicherung_niederhalter_re := TRUE;
			END_IF
			IF NOT  e_wkz_sicherung_faenger_re THEN
				sm_wkz_sicherung_faenger_re := TRUE;
				fb_state_entry.i16_next_step := FEHLER;
			END_IF
			IF NOT e_wkz_sicherung_abfallpodest_re THEN
				sm_wkz_sicherung_abfallpodest_re := TRUE;
			END_IF
		END_IF

		(*-----------------------Weiterschaltbedingungen----------------------------*)
		IF nockenschaltwerk_bestueckachse.fb.arr_spur[SP_OT]  THEN
			fb_state_entry.i16_next_step := FEHLER;
		END_IF

(*=======================================================*)
	FEHLER:
		IF fb_state_entry.E THEN
			st_ctrl_out.b_fehler := TRUE;
			fb_ton_quitt.IN := FALSE;
		END_IF

		(*-----------------------Weiterschaltbedingungen----------------------------*)
		IF st_ctrl_in.b_quitt AND NOT fb_state_entry.E THEN
			st_ctrl_out.b_fehler := FALSE;
			fb_ton_quitt.IN := TRUE;
		END_IF

		IF fb_ton_quitt.Q THEN
			fb_ton_quitt.IN := FALSE;
			fb_state_entry.i16_next_step := INIT;
		END_IF

(*=======================================================*)
	STOP:
		IF fb_state_entry.E THEN
			fb_ton_quitt.IN := FALSE;
		END_IF

		(*-----------------------Weiterschaltbedingungen----------------------------*)
		IF st_ctrl_in.b_quitt AND NOT fb_state_entry.E THEN
			fb_ton_quitt.IN := TRUE;
		END_IF

		IF fb_ton_quitt.Q THEN
			fb_ton_quitt.IN := FALSE;
			fb_state_entry.i16_next_step := INIT;
		END_IF
END_CASE

fb_state_entry(
	i16_next_step:= , 
	i16_pos:= 2,
	s_debugtext:= ,
	E=> , 
	X=> , 
	i16_step=> ,
	i16_last_step=> );

IF st_config.b_config_fertig THEN
	(* Fehlermeldungen und Betriebsmeldungen ab dem Startindex in die globalen Meldungsarrays schreiben *)
	garr_stoermeldungen[st_config.i16_meld_startindex + 0] := sm_wkz_sicherung_faenger;
	garr_stoermeldungen[st_config.i16_meld_startindex + 1] := sm_bestueckschieber_ueberwachung;
	garr_stoermeldungen[st_config.i16_meld_startindex + 2] := FALSE;
	garr_stoermeldungen[st_config.i16_meld_startindex + 3] := FALSE;
	garr_stoermeldungen[st_config.i16_meld_startindex + 4] := sm_wkz_sicherung_niederhalter_li;
	garr_stoermeldungen[st_config.i16_meld_startindex + 5] := sm_wkz_sicherung_faenger_li;
	garr_stoermeldungen[st_config.i16_meld_startindex + 6] := sm_wkz_sicherung_abfallpodest_li;
	garr_stoermeldungen[st_config.i16_meld_startindex + 7] := FALSE;
	garr_stoermeldungen[st_config.i16_meld_startindex + 8] := sm_wkz_sicherung_niederhalter_re;
	garr_stoermeldungen[st_config.i16_meld_startindex + 9] := sm_wkz_sicherung_faenger_re;
	garr_stoermeldungen[st_config.i16_meld_startindex + 10] := sm_wkz_sicherung_abfallpodest_re;
	garr_stoermeldungen[st_config.i16_meld_startindex + 11] := FALSE;
	garr_stoermeldungen[st_config.i16_meld_startindex + 12] := FALSE;
	garr_stoermeldungen[st_config.i16_meld_startindex + 13] := FALSE;
	garr_stoermeldungen[st_config.i16_meld_startindex + 14] := FALSE;
	garr_stoermeldungen[st_config.i16_meld_startindex + 15] := FALSE;
	garr_stoermeldungen[st_config.i16_meld_startindex + 16] := FALSE;
	garr_stoermeldungen[st_config.i16_meld_startindex + 17] := FALSE;
	garr_stoermeldungen[st_config.i16_meld_startindex + 18] := FALSE;
	garr_stoermeldungen[st_config.i16_meld_startindex + 19] := FALSE;
	
	garr_betriebsmeldungen[st_config.i16_meld_startindex + 0] := FALSE;
	garr_betriebsmeldungen[st_config.i16_meld_startindex + 1] := FALSE;
	garr_betriebsmeldungen[st_config.i16_meld_startindex + 2] := FALSE;
	garr_betriebsmeldungen[st_config.i16_meld_startindex + 3] := FALSE;
	garr_betriebsmeldungen[st_config.i16_meld_startindex + 4] := FALSE;
	garr_betriebsmeldungen[st_config.i16_meld_startindex + 5] := FALSE;
	garr_betriebsmeldungen[st_config.i16_meld_startindex + 6] := FALSE;
	garr_betriebsmeldungen[st_config.i16_meld_startindex + 7] := FALSE;
	garr_betriebsmeldungen[st_config.i16_meld_startindex + 8] := FALSE;
	garr_betriebsmeldungen[st_config.i16_meld_startindex + 9] := FALSE;
	garr_betriebsmeldungen[st_config.i16_meld_startindex + 10] := FALSE;
	garr_betriebsmeldungen[st_config.i16_meld_startindex + 11] := FALSE;
	garr_betriebsmeldungen[st_config.i16_meld_startindex + 12] := FALSE;
	garr_betriebsmeldungen[st_config.i16_meld_startindex + 13] := FALSE;
	garr_betriebsmeldungen[st_config.i16_meld_startindex + 14] := FALSE;
	garr_betriebsmeldungen[st_config.i16_meld_startindex + 15] := FALSE;
	garr_betriebsmeldungen[st_config.i16_meld_startindex + 16] := FALSE;
	garr_betriebsmeldungen[st_config.i16_meld_startindex + 17] := FALSE;
	garr_betriebsmeldungen[st_config.i16_meld_startindex + 18] := FALSE;
	garr_betriebsmeldungen[st_config.i16_meld_startindex + 19] := FALSE;
END_IF
END_PROGRAM

(* POU Maschine1700/Einpresskraftueberwachung/ST_Einpress_Kontroller, ST *)
PROGRAM ST_Einpress_Kontroller
VAR_INPUT
	st_config									: struct_config;
	st_ctrl_in									: struct_ctrl_in;
	lr_achsposition							: LREAL;
END_VAR
VAR_IN_OUT
	st_visu									: struct_visu;
	st_einpressen							: struct_einpresskraftueberwachung;
END_VAR
VAR_OUTPUT
	st_ctrl_out								: struct_ctrl_out;
END_VAR
VAR
	fb_ton_wz								: TON;
	fb_ton_uez								: TON;
	fb_ton_quitt								: TON;
	fb_r_trig_start								: R_TRIG;
	fb_f_trig_bestueckposzaehler				: F_TRIG;
	fb_state_entry								: ST_StateEntry;
	lr_kraft_n									: LREAL := 0.0;
	i16_pin_nr								: INT := 0;
	i16_pin_nr_alt								: INT := 0;
	i16_kraftfaktor								: INT := 0;
	sm_fehler_einpressmodus					: BOOL := FALSE;
	sm_aktkraft_groesser_maxkraft_einpressen	: BOOL := FALSE;
	sm_aktkraft_groesserr_mittelkraft_einpressen	: BOOL := FALSE;
	sm_fehler_analogwert_kraftmessdose		: BOOL := FALSE;
	sm_max_mb_ueberschritten					: BOOL := FALSE;
	sm_max_einstell_mb_ueberschritten			: BOOL := FALSE;

	a_start_messung							AT %Q* : BOOL := FALSE;
	a_messbereich_1_oder_2					AT %Q* : BOOL := FALSE;	(* MB1 = low, MB2 = high *)

	st_ausgabe								: struct_einpressausgabe;
	lr_vergleich_kraft_einpressen				: LREAL;
	lr_arr_aktuelle_kraft						: ARRAY[0..9] OF LREAL;
	lr_max_kraft_im_arr						: LREAL;
	lr_mittel_kraft_im_arr						: LREAL;
	lr_aktuelle_kraft_pin						: LREAL;
	lr_akutelle_kraft_messbereich			: LREAL;
	i										: INT;
	b_ueberwachung_gueltig					: BOOL;
END_VAR
VAR CONSTANT
	i_KRAFTFAKTOR_MB1		: INT := 200;	(* Der Kraftfaktor richtet sich nach der Messbereichskalibrierung in der Zusatzsoftware (ICAM) für den Ladungsverstärker *)
	i_KRAFTFAKTOR_MB2		: INT := 2000;
END_VAR
(* Zeiten *)
fb_ton_wz(IN:= , PT:= , Q=>  , ET=> );
fb_ton_uez(IN:= , PT:= , Q=>  , ET=> );

fb_ton_quitt(IN:= , PT:= t#100ms, Q=> , ET=> );

(* Flanken *)
fb_r_trig_start(CLK:= st_ctrl_in.b_start, Q=> );
fb_f_trig_bestueckposzaehler(CLK:= nockenschaltwerk_bestueckachse.fb.arr_spur[SP_BESTUECKSCHIEBERHUB ], Q=> );

(* Analogwert Kraftmessdose *)
kraftmessdose.fb(
	t_verzoegerung:= t#500ms,
	st_config:= kraftmessdose.fb.st_config);

(* Berechnung der aktuellen Kraft in Newton aus dem Analogwert in  Volt. *)
(* Die Normierung der Analogspannung als Kraft erfolgt mit dem Kalibrierschein der Kraftmessdose und der Software "ICAM5073" *)
(* Eingestellter Messbereich1: 0 - 200N, Messbereich2: 0 - 2000N *)
IF a_messbereich_1_oder_2 THEN
	i16_kraftfaktor := i_KRAFTFAKTOR_MB2;
ELSE
	i16_kraftfaktor := i_KRAFTFAKTOR_MB1;
END_IF

(* Behandlung Ausnahmefall Division durch 0  *)
IF kraftmessdose.fb.i16_anzeigewert_max <> 0 THEN
	lr_kraft_n := i16_kraftfaktor * kraftmessdose.fb.st_sensor.e_i16_value / kraftmessdose.fb.i16_anzeigewert_max;
END_IF

(* ===============Toplevel================ *)
IF fb_state_entry.i16_next_step > INIT AND fb_state_entry.i16_next_step < FEHLER THEN
	IF fb_state_entry.i16_next_step < STOP THEN
		IF st_ctrl_in.b_stop THEN
			fb_state_entry.i16_next_step := STOP;
		END_IF
	END_IF

	(* Fehlersignal der Kraftmessdose *)
	IF st_config.b_station_aktiv THEN
		IF kraftmessdose.fb.b_error THEN
			sm_fehler_analogwert_kraftmessdose := TRUE;
			fb_state_entry.i16_next_step := FEHLER;
		END_IF
		IF 	(NOT a_messbereich_1_oder_2 AND lr_kraft_n > i_KRAFTFAKTOR_MB1) OR
			(a_messbereich_1_oder_2 AND lr_kraft_n > i_KRAFTFAKTOR_MB2) OR
			(gst_datensatz.st_band.st_einpressen.st_einstellungen.lr_maxkraft_einpressen > i_KRAFTFAKTOR_MB2)
			THEN
				sm_max_mb_ueberschritten := TRUE;
				fb_state_entry.i16_next_step := FEHLER;
		END_IF
		IF gst_datensatz.st_band.st_einpressen.st_einstellungen.lr_maxkraft_einpressen > i_KRAFTFAKTOR_MB2 THEN
			sm_max_einstell_mb_ueberschritten := TRUE;
			fb_state_entry.i16_next_step := FEHLER;
		END_IF
	END_IF
END_IF

(* ======================================Schrittkette======================================== *)
fb_state_entry(
	i16_next_step:= ,
	i16_pos:= 1,
	s_debugtext:= ,
	E=> ,
	X=> ,
	i16_step=> ,
	i16_last_step=> );

CASE fb_state_entry.i16_step OF
(*=======================================================*)
	INIT_OBJ:
		IF st_config.b_config_fertig THEN
			a_messbereich_1_oder_2 := FALSE;
			fb_state_entry.i16_next_step := INIT;
		END_IF

(*=======================================================*)
	INIT:
		IF fb_state_entry.E THEN
			fb_ton_wz.IN := FALSE;
			fb_ton_uez.IN := FALSE;
			fb_ton_quitt.IN := FALSE;
			st_ctrl_out.b_fehler := FALSE;
			st_ctrl_out.b_bereit := FALSE;
			st_ctrl_out.b_fertig := FALSE;
			a_start_messung := FALSE;
			b_ueberwachung_gueltig := FALSE;
			i16_pin_nr := 0;
			sm_fehler_einpressmodus := FALSE;
			sm_aktkraft_groesser_maxkraft_einpressen := FALSE;
			sm_aktkraft_groesserr_mittelkraft_einpressen := FALSE;
			sm_fehler_analogwert_kraftmessdose := FALSE;
			sm_max_mb_ueberschritten := FALSE;
			sm_max_einstell_mb_ueberschritten := FALSE;
			(*Löschen der gesammelten Kräfte der letzten zehn Hübe*)
			FOR i := 0 TO 9 DO
				lr_arr_aktuelle_kraft[i] := 0;
			END_FOR

		END_IF

		(*-----------------------Weiterschaltbedingungen----------------------------*)
		IF st_ctrl_in.b_init THEN
			fb_state_entry.i16_next_step := BEREIT;
		END_IF

(*=======================================================*)
	BEREIT:
		IF fb_state_entry.E THEN
			st_ctrl_out.b_bereit := TRUE;
			st_ctrl_out.b_fertig := TRUE;
			i16_pin_nr := 0;
			i16_pin_nr_alt := 0;
		END_IF

		(*-----------------------Weiterschaltbedingungen----------------------------*)
		IF st_ctrl_in.b_start THEN
			fb_state_entry.i16_next_step := 110;
		END_IF

(*=======================================================*)
	110:	(* Kraftmessung starten *)
		IF fb_state_entry.E THEN
			st_ctrl_out.b_fertig := FALSE;
			a_start_messung := TRUE;
			st_ausgabe.st_ergebnisse.lr_maxkraft_einpressen := 0;
			st_ausgabe.st_ergebnisse.lr_maxkraft_einpres_proHub:=0;
			st_ausgabe.st_ergebnisse.lr_ueberlaufkraft := 0;
			lr_aktuelle_kraft_pin := 0;
			lr_akutelle_kraft_messbereich := 0;
		END_IF

		(* Hochzählen mit der Anzahl der bestückten Pins *)
		IF fb_f_trig_bestueckposzaehler.Q THEN
			i16_pin_nr := i16_pin_nr +1;
		END_IF

		(*aktuell höchste Kraft wird sich gemerkt*)
		IF  lr_kraft_n > lr_aktuelle_kraft_pin THEN
			lr_aktuelle_kraft_pin := lr_kraft_n;
			lr_akutelle_kraft_messbereich := lr_kraft_n;
		END_IF

		(*Bei jedem neuen Pin wird die höchste gemessene Kraft in ein Array geschrieben und die älteste von den letzten 10
		wird gelöscht*)
		IF i16_pin_nr_alt <> i16_pin_nr AND ST_Virtuelle_Masterachse.i16_bestueckachse_cam_table_id = 5 THEN
			FOR i:=9 TO 1 BY -1 DO
				lr_arr_aktuelle_kraft[i]:=lr_arr_aktuelle_kraft[i-1];
			END_FOR
			lr_arr_aktuelle_kraft[0] := lr_aktuelle_kraft_pin;
			lr_aktuelle_kraft_pin := 0;
			i16_pin_nr_alt := i16_pin_nr;
		END_IF

		(*Überprüfung, ob das Array komplett mit Werten befüllt ist*)
		FOR i := 0 TO 9 DO
			IF lr_arr_aktuelle_kraft[i] = 0 THEN
				b_ueberwachung_gueltig := FALSE;
				EXIT;
			ELSE
				b_ueberwachung_gueltig := TRUE;
			END_IF
		END_FOR

		(*Auswahl Auswertemodus*)
		CASE st_einpressen.st_einstellungen.enu_modus OF

			KEIN_MODUS:	(* Kraftübwerachung ausgeschalten *)
					;
			F_MAXWERT:	(* Einpressen mit Überwachung auf den Maximalwert *)

				IF b_ueberwachung_gueltig THEN
					lr_max_kraft_im_arr := 0;
					(*Maximalkraft im Array wird gesucht*)
					FOR i := 0 TO 9 DO
						IF  lr_arr_aktuelle_kraft[i] > lr_max_kraft_im_arr THEN
							lr_max_kraft_im_arr := lr_arr_aktuelle_kraft[i];
						END_IF
					END_FOR

					(* nur bei voller Drehzahl und normalen Bestückbild mit ermittelter Kraft prüfen*)
					IF ST_TippTasten.i16_akt_stufe = 9 AND (FIND(gst_datensatz.st_md.s_aktuelle_artikelnummer,'ruef') = 0		(*es wird nur auf ruef abgefragt, weil das P groß oder klein sein kann*)
						 AND FIND(gst_datensatz.st_md.s_aktuelle_artikelnummer,'erth') = 0) THEN
						lr_vergleich_kraft_einpressen:=lr_max_kraft_im_arr;
					ELSE
						lr_vergleich_kraft_einpressen:=800;
					END_IF

					(* Fehlerfall: Ermittelte Maximalkraft überschritten nur im Automatik Betrieb *)
					IF  gi16_betriebsart = AUTO AND lr_kraft_n > lr_vergleich_kraft_einpressen + st_einpressen.st_einstellungen.lr_delta_kraft THEN
						st_einpressen.st_einstellungen.lr_maxkraft_einpressen := lr_kraft_n;
						st_ausgabe.st_ergebnisse.lr_maxkraft_einpressen:=lr_kraft_n;
						sm_aktkraft_groesser_maxkraft_einpressen := TRUE;
						fb_state_entry.i16_next_step := FEHLER;
					END_IF
				END_IF


			F_MITTELWERT:	(* Einpressen mit Überwachung auf den Mittelwert *)

				IF b_ueberwachung_gueltig THEN
					(*Kraft im Array wird aufaddiert*)
					FOR i := 0 TO 9 DO
						lr_mittel_kraft_im_arr := lr_mittel_kraft_im_arr + lr_arr_aktuelle_kraft[i];
					END_FOR
					(*Mittelwert der Kräfte im Array wird gebildet*)
					lr_mittel_kraft_im_arr := lr_mittel_kraft_im_arr / 10;

					(* nur bei voller Drehzahl und normalen Bestückbild mit ermittelter Kraft prüfen*)
					IF ST_TippTasten.i16_akt_stufe = 9 AND (FIND(gst_datensatz.st_md.s_aktuelle_artikelnummer,'ruef') = 0			(*es wird nur auf ruef abgefragt, weil das P groß oder klein sein kann*)
						AND FIND(gst_datensatz.st_md.s_aktuelle_artikelnummer,'erth') = 0) THEN
						lr_vergleich_kraft_einpressen:=lr_mittel_kraft_im_arr;
					ELSE
						lr_vergleich_kraft_einpressen:=800;
					END_IF

					(* Fehlerfall: Ermittelte Maximalkraft überschritten nur im Automatik Betrieb *)
					IF  gi16_betriebsart = AUTO AND lr_kraft_n > lr_vergleich_kraft_einpressen + st_einpressen.st_einstellungen.lr_delta_kraft THEN
						sm_aktkraft_groesserr_mittelkraft_einpressen := TRUE;
						st_einpressen.st_einstellungen.lr_maxkraft_einpressen := lr_kraft_n;
						st_ausgabe.st_ergebnisse.lr_maxkraft_einpressen:=lr_kraft_n;
						fb_state_entry.i16_next_step := FEHLER;
					END_IF
				END_IF
		END_CASE

		(* Manuelle Messbereichsumschaltung anhand des Einstellwertes für Maximalkraft beim Einpressen. *)
		IF gst_datensatz.st_band.st_einpressen.st_einstellungen.lr_maxkraft_einpressen > (i_KRAFTFAKTOR_MB1 * 0.75) THEN
			a_messbereich_1_oder_2 := TRUE;
		ELSE
			(* Automatische Messbereichsumschaltung, wenn die maximale Einpresskraft 75% des Messbereichsendwertes überschreitet. *)
			IF lr_akutelle_kraft_messbereich > (i_KRAFTFAKTOR_MB1 * 0.75) THEN
				a_messbereich_1_oder_2 := TRUE;
			END_IF
		END_IF

		(*-----------------------Weiterschaltbedingungen----------------------------*)
		IF NOT st_ctrl_in.b_start THEN
			(* Messbereichsanpassung nur, wenn die Krafteinstellung für maximale Einpresskraft es erlaubt. *)
			IF gst_datensatz.st_band.st_einpressen.st_einstellungen.lr_maxkraft_einpressen < (i_KRAFTFAKTOR_MB1 * 0.75) THEN
				(* Automatische Messbereichsumschaltung, wenn die maximale Einpresskraft 50% des Messbereichsendwertes unterschreitet. *)
				IF lr_akutelle_kraft_messbereich < (i_KRAFTFAKTOR_MB1 * 0.5) THEN
					a_messbereich_1_oder_2 := FALSE;
				END_IF
			END_IF
			a_start_messung := FALSE;
			fb_state_entry.i16_next_step := BEREIT;
		END_IF

(*=======================================================*)
	FEHLER:
		IF fb_state_entry.E THEN
			st_ctrl_out.b_fehler := TRUE;
			fb_ton_quitt.IN := FALSE;
		END_IF

		(* Aufzeichnen der Überlaufkraft nach einem Einpressfehler *)
		IF  lr_kraft_n > st_ausgabe.st_ergebnisse.lr_ueberlaufkraft THEN
			st_ausgabe.st_ergebnisse.lr_ueberlaufkraft := lr_kraft_n;
		END_IF

		(*-----------------------Weiterschaltbedingungen----------------------------*)
		IF st_ctrl_in.b_quitt AND NOT fb_state_entry.E THEN
			st_ctrl_out.b_fehler := FALSE;
			fb_ton_quitt.IN := TRUE;
		END_IF

		IF fb_ton_quitt.Q THEN
			fb_ton_quitt.IN := FALSE;
			fb_state_entry.i16_next_step := INIT;
		END_IF

(*=======================================================*)
	STOP:
		IF fb_state_entry.E THEN
			fb_ton_quitt.IN := FALSE;
		END_IF

		(*-----------------------Weiterschaltbedingungen----------------------------*)
		IF st_ctrl_in.b_quitt AND NOT fb_state_entry.E THEN
			fb_ton_quitt.IN := TRUE;
		END_IF

		IF fb_ton_quitt.Q THEN
			fb_ton_quitt.IN := FALSE;
			fb_state_entry.i16_next_step := INIT;
		END_IF
END_CASE

fb_state_entry(
	i16_next_step:= ,
	i16_pos:= 2,
	s_debugtext:= ,
	E=> ,
	X=> ,
	i16_step=> ,
	i16_last_step=> );

(* Fehlermeldungen und Betriebsmeldungen ab dem Startindex in die globalen Meldungsarrays schreiben *)
garr_stoermeldungen[st_config.i16_meld_startindex + 0] := sm_fehler_einpressmodus;
garr_stoermeldungen[st_config.i16_meld_startindex + 1] := sm_aktkraft_groesser_maxkraft_einpressen;
garr_stoermeldungen[st_config.i16_meld_startindex + 2] := sm_aktkraft_groesserr_mittelkraft_einpressen;
garr_stoermeldungen[st_config.i16_meld_startindex + 3] := sm_fehler_analogwert_kraftmessdose;
garr_stoermeldungen[st_config.i16_meld_startindex + 4] := sm_max_mb_ueberschritten;
garr_stoermeldungen[st_config.i16_meld_startindex + 5] := sm_max_einstell_mb_ueberschritten;
garr_stoermeldungen[st_config.i16_meld_startindex + 6] := FALSE;
garr_stoermeldungen[st_config.i16_meld_startindex + 7] := FALSE;
garr_stoermeldungen[st_config.i16_meld_startindex + 8] := FALSE;
garr_stoermeldungen[st_config.i16_meld_startindex + 9] := FALSE;
garr_stoermeldungen[st_config.i16_meld_startindex + 10] := FALSE;
garr_stoermeldungen[st_config.i16_meld_startindex + 11] := FALSE;
garr_stoermeldungen[st_config.i16_meld_startindex + 12] := FALSE;
garr_stoermeldungen[st_config.i16_meld_startindex + 13] := FALSE;
garr_stoermeldungen[st_config.i16_meld_startindex + 14] := FALSE;
garr_stoermeldungen[st_config.i16_meld_startindex + 15] := FALSE;
garr_stoermeldungen[st_config.i16_meld_startindex + 16] := FALSE;
garr_stoermeldungen[st_config.i16_meld_startindex + 17] := FALSE;
garr_stoermeldungen[st_config.i16_meld_startindex + 18] := FALSE;
garr_stoermeldungen[st_config.i16_meld_startindex + 19] := FALSE;

garr_betriebsmeldungen[st_config.i16_meld_startindex + 0] := FALSE;
garr_betriebsmeldungen[st_config.i16_meld_startindex + 1] := FALSE;
garr_betriebsmeldungen[st_config.i16_meld_startindex + 2] := FALSE;
garr_betriebsmeldungen[st_config.i16_meld_startindex + 3] := FALSE;
garr_betriebsmeldungen[st_config.i16_meld_startindex + 4] := FALSE;
garr_betriebsmeldungen[st_config.i16_meld_startindex + 5] := FALSE;
garr_betriebsmeldungen[st_config.i16_meld_startindex + 6] := FALSE;
garr_betriebsmeldungen[st_config.i16_meld_startindex + 7] := FALSE;
garr_betriebsmeldungen[st_config.i16_meld_startindex + 8] := FALSE;
garr_betriebsmeldungen[st_config.i16_meld_startindex + 9] := FALSE;
garr_betriebsmeldungen[st_config.i16_meld_startindex + 10] := FALSE;
garr_betriebsmeldungen[st_config.i16_meld_startindex + 11] := FALSE;
garr_betriebsmeldungen[st_config.i16_meld_startindex + 12] := FALSE;
garr_betriebsmeldungen[st_config.i16_meld_startindex + 13] := FALSE;
garr_betriebsmeldungen[st_config.i16_meld_startindex + 14] := FALSE;
garr_betriebsmeldungen[st_config.i16_meld_startindex + 15] := FALSE;
garr_betriebsmeldungen[st_config.i16_meld_startindex + 16] := FALSE;
garr_betriebsmeldungen[st_config.i16_meld_startindex + 17] := FALSE;
garr_betriebsmeldungen[st_config.i16_meld_startindex + 18] := FALSE;
garr_betriebsmeldungen[st_config.i16_meld_startindex + 19] := FALSE;
END_PROGRAM

(* POU Maschine1700/Band/ST_Bandeinzug_Kontroller_1700, ST *)
PROGRAM ST_Bandeinzug_Kontroller_1700
VAR_INPUT
	st_config						: struct_config;
	st_ctrl_in						: struct_ctrl_in;
END_VAR
VAR_IN_OUT
	st_visu						: struct_visu;
END_VAR
VAR_OUTPUT
	st_ctrl_out					: struct_ctrl_out;
END_VAR
VAR
	fb_ton_wz					: TON;
	fb_ton_uez					: TON;
	fb_ton_quitt					: TON;
	fb_state_entry					: ST_StateEntry;
	b_einzug_stop				: BOOL := FALSE;

	fb_r_trig_vorschubkontrolle		: R_TRIG;
	fb_f_trig_vorschubkontrolle		: F_TRIG;
	fb_r_trig_nocke_einzug			: R_TRIG;
	fb_f_trig_nocke_einzug			: F_TRIG;
	b_hm_pos_flanke_vorschub	: BOOL := FALSE;
	b_hm_neg_flanke_vorschub	: BOOL := FALSE;
	sm_fehler_bandvorschub		: BOOL := FALSE;
	sm_keine_busverbindung	: BOOL := FALSE;

	e_wc_state					AT %I* : BOOL;	(* 0=Data valid, 1=Data invalid *)
	e_gls_bandvorschubkontrolle	AT %I* : BOOL;
END_VAR
(* Zeiten *)
fb_ton_wz(IN:= , PT:= , Q=>  , ET=> );
fb_ton_uez(IN:= , PT:= , Q=>  , ET=> );
fb_ton_quitt(IN:= , PT:= t#100ms, Q=> , ET=> );

(* Flanken *)
fb_f_trig_vorschubkontrolle(CLK:= e_gls_bandvorschubkontrolle, Q=> );
fb_r_trig_vorschubkontrolle(CLK:= e_gls_bandvorschubkontrolle, Q=> );
fb_f_trig_nocke_einzug(CLK:= nockenschaltwerk_bestueckachse.fb.arr_spur[SP_PNEUMATIKBANDEINZUG_GLS], Q=> );
fb_r_trig_nocke_einzug(CLK:= nockenschaltwerk_bestueckachse.fb.arr_spur[SP_PNEUMATIKBANDEINZUG_GLS], Q=> );

(* Toplevel *)
IF fb_state_entry.i16_next_step > INIT AND fb_state_entry.i16_next_step < FEHLER THEN
	IF fb_state_entry.i16_next_step < STOP THEN
		IF st_ctrl_in.b_stop THEN
			fb_state_entry.i16_next_step := STOP;
		END_IF
	END_IF
	(* Allgemeine Fehler *)
	IF	NOT gst_datensatz.st_md.b_wt_transport_simulation AND
		(zyl_bandfaenger.st_ctrl.out.b_fehler OR
		zyl_bandklemmen.st_ctrl.out.b_fehler)
		 THEN
			fb_state_entry.i16_next_step := FEHLER;

	(* Zylinder im Handbetrieb *)
	ELSIF	 gi16_betriebsart = HAND AND (
			(st_visu.st_zyl.i16_nr_zyl_im_handbetrieb = zyl_bandfaenger.fb.st_config.i16_identnummer) OR
			(st_visu.st_zyl.i16_nr_zyl_im_handbetrieb = zyl_bandklemmen.fb.st_config.i16_identnummer) )
			THEN
			fb_state_entry.i16_next_step := FEHLER;
	END_IF
END_IF

(* ======================================Schrittkette======================================== *)
fb_state_entry(
	i16_next_step:= , 
	i16_pos:= 1,
	s_debugtext:= ,
	E=> ,
	X=> , 
	i16_step=> ,
	i16_last_step=> );

CASE fb_state_entry.i16_step OF
(*=======================================================*)
	INIT_OBJ:
		IF st_config.b_config_fertig THEN
			fb_state_entry.i16_next_step := INIT;
		END_IF

(*=======================================================*)
	INIT:
		IF fb_state_entry.E THEN
			fb_ton_wz.IN := FALSE;
			fb_ton_uez.IN := FALSE;
			fb_ton_quitt.IN := FALSE;
			st_ctrl_out.b_fehler := FALSE;
			st_ctrl_out.b_bereit := FALSE;
			st_ctrl_out.b_fertig := FALSE;
			zyl_bandfaenger.st_ctrl.in.b_ausfahren := FALSE;
			zyl_bandfaenger.st_ctrl.in.b_einfahren := FALSE;
			 zyl_bandklemmen.st_ctrl.in.b_ausfahren := FALSE;
			 zyl_bandklemmen.st_ctrl.in.b_einfahren := FALSE;
			sm_fehler_bandvorschub := FALSE;
			sm_keine_busverbindung := FALSE;
		END_IF

		(*-----------------------Weiterschaltbedingungen----------------------------*)
		IF st_ctrl_in.b_init THEN
			zyl_bandfaenger.st_ctrl.in.b_quittieren := FALSE;
			 zyl_bandklemmen.st_ctrl.in.b_quittieren := FALSE;
			IF gst_datensatz.st_md.b_wt_transport_simulation THEN
				fb_state_entry.i16_next_step := BEREIT;
			ELSE
				(*fb_state_entry.i16_next_step := 20; Bei nächster TSM-Änderung bitte aktivieren*)
				fb_state_entry.i16_next_step := BEREIT;
			END_IF
		END_IF

(*=======================================================*)
	20: (* Prüfe, ob Busverbindung vorhanden ist *)

		(*-----------------------Weiterschaltbedingungen----------------------------*)
		IF e_wc_state THEN	(* Prüfe Busverbindung ( 0=Data valid, 1=Data invalid )*)
			sm_keine_busverbindung := TRUE;
			fb_state_entry.i16_next_step := FEHLER;
		ELSE
			fb_state_entry.i16_next_step := BEREIT;
		END_IF

(*=======================================================*)
	BEREIT:
		IF fb_state_entry.E THEN
			st_ctrl_out.b_bereit := TRUE;
		END_IF

		(*-----------------------Weiterschaltbedingungen----------------------------*)
		CASE gst_datensatz.st_wkz.i16_typ_bandeinzug OF
			BANDWECHSLER_V2:
				(* Versuchsablauf zum mehrfach Biegen eines Bandes *)
				(* Die Anzahl der Werkzeughübe zum Biegen wird durch das Bestückprogramm bestimmt *)
				IF b_einzug_stop AND nockenschaltwerk_bestueckachse.fb.arr_spur[SP_OT] THEN
					fb_state_entry.i16_next_step := 500;
				ELSE
					fb_state_entry.i16_next_step := 200;
				END_IF
			SERVO:
				;
		END_CASE;

(*===========================Bandvorschub mit GLS-Kontrolle============================*)
	200:	(* Warte auf Vorschubnocke  und Freigabe von der Bestückachse *)
		(* Die Freigabe erfolgt nur im normalen Produktionsablauf; nicht bei Bandwechsel, Einfädeln, ... da hier keine Überwachung erfolgen soll. *)

		(*-----------------------Weiterschaltbedingungen----------------------------*)
		IF fb_r_trig_nocke_einzug.Q AND gi16_betriebsart <> HAND AND st_ctrl_in.b_freigabe THEN
			b_hm_pos_flanke_vorschub := FALSE;
			b_hm_neg_flanke_vorschub := FALSE;
			fb_state_entry.i16_next_step := 210;
		END_IF

(*=======================================================*)
	210:	(* Band wird vorgeschoben *)
		(* Vorschubkontrolle durch positive Flanke *)
		IF fb_r_trig_vorschubkontrolle.Q THEN
			b_hm_pos_flanke_vorschub := TRUE;
		END_IF
		(* Vorschubkontrolle durch negative Flanke *)
		IF fb_f_trig_vorschubkontrolle.Q THEN
			b_hm_neg_flanke_vorschub := TRUE;
		END_IF

		(* bei abgeschalteten Nocken *)
		IF	NOT gst_datensatz.st_wkz.nockenschaltwerk_bestueckachse.arr_nocken[NO_PNEUMATIKBANDEINZUG_GLS].b_camvalid THEN
			b_hm_neg_flanke_vorschub := TRUE;
			b_hm_pos_flanke_vorschub := TRUE;
		END_IF
		(*-----------------------Weiterschaltbedingungen----------------------------*)
		IF fb_f_trig_nocke_einzug.Q THEN
			IF b_hm_pos_flanke_vorschub AND b_hm_neg_flanke_vorschub THEN
				fb_state_entry.i16_next_step := 200;
			ELSE
				sm_fehler_bandvorschub := TRUE;
				fb_state_entry.i16_next_step := FEHLER;
			END_IF
		ELSIF gi16_betriebsart = HAND OR NOT st_ctrl_in.b_freigabe THEN
			fb_state_entry.i16_next_step := 200;
		END_IF

(*=======================================================*)
	500:	(* Nocken deaktivieren und Bandfänger deaktivieren/einfahren sowie Bandklemmen ausfahren*)
		IF fb_state_entry.E THEN
			CASE gst_datensatz.st_wkz.i16_typ_bandeinzug OF

				BANDWECHSLER_V2:
					(* Bandwechsler V2 ohne Sensoren und anderen Zylindern *)
					gst_datensatz.st_wkz.nockenschaltwerk_bestueckachse.arr_nocken[NO_BW_BANDFAENGER_BAWEV2_EINFAHREN].b_camvalid := FALSE;
					gst_datensatz.st_wkz.nockenschaltwerk_bestueckachse.arr_nocken[NO_BW_BANDFAENGER_BAWEV2_AUSFAHREN].b_camvalid := FALSE;
					gst_datensatz.st_wkz.nockenschaltwerk_bestueckachse.arr_nocken[NO_BW_BANDKLEMMEN_BAWEV2_EINFAHREN].b_camvalid := FALSE;
					gst_datensatz.st_wkz.nockenschaltwerk_bestueckachse.arr_nocken[NO_BW_BANDKLEMMEN_BAWEV2_AUSFAHREN].b_camvalid := FALSE;
				SERVO:
					;
			END_CASE;

			zyl_bandfaenger.fb.b_no_gesteuert_im_norm_betrieb := TRUE;
			zyl_bandklemmen.fb.b_no_gesteuert_im_norm_betrieb := TRUE;
			(* Zylinder einfahren *)
			zyl_bandfaenger.st_ctrl.in.b_einfahren := TRUE;
			zyl_bandklemmen.st_ctrl.in.b_ausfahren := TRUE;
		END_IF

		(*-----------------------Weiterschaltbedingungen----------------------------*)
		IF zyl_bandfaenger.st_ctrl.out.b_eingefahren AND zyl_bandklemmen.st_ctrl.out.b_ausgefahren AND gb_ba_auto_kontroller THEN
			zyl_bandfaenger.st_ctrl.in.b_einfahren := FALSE;
			zyl_bandklemmen.st_ctrl.in.b_ausfahren := FALSE;
			fb_state_entry.i16_next_step := 510;
		END_IF

(*=======================================================*)
	510:
		IF fb_state_entry.E THEN
			;
		END_IF

		(*-----------------------Weiterschaltbedingungen----------------------------*)
		IF NOT b_einzug_stop THEN
			(* Bandwechsler V1 *)
			gst_datensatz.st_wkz.nockenschaltwerk_bestueckachse.arr_nocken[NO_BW_BANDFAENGER_EINFAHREN].b_camvalid := TRUE;
			gst_datensatz.st_wkz.nockenschaltwerk_bestueckachse.arr_nocken[NO_BW_BANDFAENGER_AUSFAHREN].b_camvalid := TRUE;
			gst_datensatz.st_wkz.nockenschaltwerk_bestueckachse.arr_nocken[NO_UW_BANDFAENGER_EINFAHREN].b_camvalid := TRUE;
			gst_datensatz.st_wkz.nockenschaltwerk_bestueckachse.arr_nocken[NO_UW_BANDFAENGER_AUSFAHREN].b_camvalid := TRUE;
			gst_datensatz.st_wkz.nockenschaltwerk_bestueckachse.arr_nocken[NO_BW_BANDKLEMMEN_EINFAHREN].b_camvalid := TRUE;
			gst_datensatz.st_wkz.nockenschaltwerk_bestueckachse.arr_nocken[NO_BW_BANDKLEMMEN_AUSFAHREN].b_camvalid := TRUE;
			gst_datensatz.st_wkz.nockenschaltwerk_bestueckachse.arr_nocken[NO_UW_BANDKLEMMEN_EINFAHREN].b_camvalid := TRUE;
			gst_datensatz.st_wkz.nockenschaltwerk_bestueckachse.arr_nocken[NO_UW_BANDKLEMMEN_AUSFAHREN].b_camvalid := TRUE;
			(* Bandwechsler V2 ohne Sensoren und anderen Zylindern *)
			gst_datensatz.st_wkz.nockenschaltwerk_bestueckachse.arr_nocken[NO_BW_BANDFAENGER_BAWEV2_EINFAHREN].b_camvalid := TRUE;
			gst_datensatz.st_wkz.nockenschaltwerk_bestueckachse.arr_nocken[NO_BW_BANDFAENGER_BAWEV2_AUSFAHREN].b_camvalid := TRUE;
			gst_datensatz.st_wkz.nockenschaltwerk_bestueckachse.arr_nocken[NO_BW_BANDKLEMMEN_BAWEV2_EINFAHREN].b_camvalid := TRUE;
			gst_datensatz.st_wkz.nockenschaltwerk_bestueckachse.arr_nocken[NO_BW_BANDKLEMMEN_BAWEV2_AUSFAHREN].b_camvalid := TRUE;

			zyl_bandfaenger.fb.b_no_gesteuert_im_norm_betrieb := FALSE;
			zyl_bandklemmen.fb.b_no_gesteuert_im_norm_betrieb := FALSE;
			fb_state_entry.i16_next_step := BEREIT;
		END_IF

(*=======================================================*)
	FEHLER:
		IF fb_state_entry.E THEN
			st_ctrl_out.b_fehler := TRUE;
			fb_ton_quitt.IN := FALSE;
			zyl_bandfaenger.st_ctrl.in.b_quittieren := FALSE;
			zyl_bandklemmen.st_ctrl.in.b_quittieren := FALSE;
		END_IF

		(*-----------------------Weiterschaltbedingungen----------------------------*)
		IF st_ctrl_in.b_quitt AND NOT fb_state_entry.E THEN
			st_ctrl_out.b_fehler := FALSE;
			zyl_bandfaenger.st_ctrl.in.b_quittieren := TRUE;
			zyl_bandklemmen.st_ctrl.in.b_quittieren := TRUE;
			fb_ton_quitt.IN := TRUE;
		END_IF

		IF fb_ton_quitt.Q THEN
			fb_ton_quitt.IN := FALSE;
			fb_state_entry.i16_next_step := INIT;
		END_IF

(*=======================================================*)
	STOP:
		IF fb_state_entry.E THEN
			fb_ton_quitt.IN := FALSE;
			zyl_bandfaenger.st_ctrl.in.b_quittieren := FALSE;
			zyl_bandklemmen.st_ctrl.in.b_quittieren := FALSE;
		END_IF

		(*-----------------------Weiterschaltbedingungen----------------------------*)
		IF st_ctrl_in.b_quitt AND NOT fb_state_entry.E THEN
			fb_ton_quitt.IN := TRUE;
			zyl_bandfaenger.st_ctrl.in.b_quittieren := TRUE;
			zyl_bandklemmen.st_ctrl.in.b_quittieren := TRUE;
		END_IF

		IF fb_ton_quitt.Q THEN
			fb_ton_quitt.IN := FALSE;
			fb_state_entry.i16_next_step := INIT;
		END_IF
END_CASE

fb_state_entry(
	i16_next_step:= , 
	i16_pos:= 2,
	s_debugtext:= ,
	E=> , 
	X=> , 
	i16_step=> ,
	i16_last_step=> );

IF st_config.b_config_fertig THEN
	(* Fehlermeldungen und Betriebsmeldungen ab dem Startindex in die globalen Meldungsarrays schreiben *)
	garr_stoermeldungen[st_config.i16_meld_startindex + 0] := sm_fehler_bandvorschub;
	garr_stoermeldungen[st_config.i16_meld_startindex + 1] := FALSE;(* belegt  durch Bandeinzugskontroller 1720 *)
	garr_stoermeldungen[st_config.i16_meld_startindex + 2] := FALSE;(* belegt  durch Bandeinzugskontroller 1720 *)
	garr_stoermeldungen[st_config.i16_meld_startindex + 3] := sm_keine_busverbindung;
	garr_stoermeldungen[st_config.i16_meld_startindex + 4] := FALSE;
	garr_stoermeldungen[st_config.i16_meld_startindex + 5] := FALSE;
	garr_stoermeldungen[st_config.i16_meld_startindex + 6] := FALSE;
	garr_stoermeldungen[st_config.i16_meld_startindex + 7] := FALSE;
	garr_stoermeldungen[st_config.i16_meld_startindex + 8] := FALSE;
	garr_stoermeldungen[st_config.i16_meld_startindex + 9] := FALSE;
	garr_stoermeldungen[st_config.i16_meld_startindex + 10] := FALSE;
	garr_stoermeldungen[st_config.i16_meld_startindex + 11] := FALSE;
	garr_stoermeldungen[st_config.i16_meld_startindex + 12] := FALSE;
	garr_stoermeldungen[st_config.i16_meld_startindex + 13] := FALSE;
	garr_stoermeldungen[st_config.i16_meld_startindex + 14] := FALSE;
	garr_stoermeldungen[st_config.i16_meld_startindex + 15] := FALSE;
	garr_stoermeldungen[st_config.i16_meld_startindex + 16] := FALSE;
	garr_stoermeldungen[st_config.i16_meld_startindex + 17] := FALSE;
	garr_stoermeldungen[st_config.i16_meld_startindex + 18] := FALSE;
	garr_stoermeldungen[st_config.i16_meld_startindex + 19] := FALSE;
	
	garr_betriebsmeldungen[st_config.i16_meld_startindex + 0] := FALSE;
	garr_betriebsmeldungen[st_config.i16_meld_startindex + 1] := FALSE;
	garr_betriebsmeldungen[st_config.i16_meld_startindex + 2] := FALSE;
	garr_betriebsmeldungen[st_config.i16_meld_startindex + 3] := FALSE;
	garr_betriebsmeldungen[st_config.i16_meld_startindex + 4] := FALSE;
	garr_betriebsmeldungen[st_config.i16_meld_startindex + 5] := FALSE;
	garr_betriebsmeldungen[st_config.i16_meld_startindex + 6] := FALSE;
	garr_betriebsmeldungen[st_config.i16_meld_startindex + 7] := FALSE;
	garr_betriebsmeldungen[st_config.i16_meld_startindex + 8] := FALSE;
	garr_betriebsmeldungen[st_config.i16_meld_startindex + 9] := FALSE;
	garr_betriebsmeldungen[st_config.i16_meld_startindex + 10] := FALSE;
	garr_betriebsmeldungen[st_config.i16_meld_startindex + 11] := FALSE;
	garr_betriebsmeldungen[st_config.i16_meld_startindex + 12] := FALSE;
	garr_betriebsmeldungen[st_config.i16_meld_startindex + 13] := FALSE;
	garr_betriebsmeldungen[st_config.i16_meld_startindex + 14] := FALSE;
	garr_betriebsmeldungen[st_config.i16_meld_startindex + 15] := FALSE;
	garr_betriebsmeldungen[st_config.i16_meld_startindex + 16] := FALSE;
	garr_betriebsmeldungen[st_config.i16_meld_startindex + 17] := FALSE;
	garr_betriebsmeldungen[st_config.i16_meld_startindex + 18] := FALSE;
	garr_betriebsmeldungen[st_config.i16_meld_startindex + 19] := FALSE;
END_IF
END_PROGRAM

(* POU Gemeinsamkeiten17xx/Zylinder/ST_Zylinder_Fast, ST *)
PROGRAM ST_Zylinder_Fast
VAR
END_VAR
(* Zylinderaufrufe *)
CASE gst_datensatz.st_md.i16_typ_zelle OF
	KEINE_ZELLE:
		;

	BESTUECKZELLE_1700:
		ST_Datainit_Fast_Zylinder();

		CASE gst_datensatz.st_wkz.i16_typ_bandeinzug OF
			KEIN_EINZUG:
				;

			STANDARD_2FACH_V2:
				;

				BANDWECHSLER_V2:
				zyl_bandfaenger.fb.st_config.b_aktiv := NOT gst_datensatz.st_md.b_wt_transport_simulation;
				zyl_bandfaenger.fb(
					st_config:= ,
					e_druckwaechter:= ST_Betriebsfreigaben.e_druckwaechter,
					i16_betriebsart:= gi16_betriebsart,
					b_no_gesteuert_im_norm_betrieb:= ,
					b_direkttaste_ausfahren:= ,
					b_direkttaste_mittefahren:= ,
					b_direkttaste_einfahren	:= ,
					st_ctrl_in:= zyl_bandfaenger.st_ctrl.in,
					b_masterachse_hand_dialog_aktiv:= ST_Bestueckachse.b_hand_dialog_aktiv,
					st_visu:= visu.st_zyl,
					bw_nocken_zylinder_einfahren := nockenschaltwerk_bestueckachse.fb.arr_spur[SP_BW_BANDFAENGER_BAWEV2_EINFAHREN],
					bw_nocken_zylinder_ausfahren := nockenschaltwerk_bestueckachse.fb.arr_spur[SP_BW_BANDFAENGER_BAWEV2_AUSFAHREN],
					uw_nocken_zylinder_einfahren := ,
					uw_nocken_zylinder_ausfahren := ,
					st_ctrl_out=> zyl_bandfaenger.st_ctrl.out,
					a_ventil_einfahren=> a_zyl_faenger_einfahren,
					a_ventil_ausfahren=> );
		
				zyl_bandklemmen.fb.st_config.b_aktiv := NOT gst_datensatz.st_md.b_wt_transport_simulation;
				zyl_bandklemmen.fb(
					st_config:= ,
					e_druckwaechter:= ST_Betriebsfreigaben.e_druckwaechter,
					i16_betriebsart:= gi16_betriebsart,
					b_no_gesteuert_im_norm_betrieb:= ,
					b_direkttaste_ausfahren:= ,
					b_direkttaste_mittefahren:= ,
					b_direkttaste_einfahren	:= ,
					st_ctrl_in:= zyl_bandklemmen.st_ctrl.in,
					b_masterachse_hand_dialog_aktiv:= ST_Bestueckachse.b_hand_dialog_aktiv,
					st_visu:= visu.st_zyl,
					bw_nocken_zylinder_einfahren := nockenschaltwerk_bestueckachse.fb.arr_spur[SP_BW_BANDKLEMMEN_BAWEV2_EINFAHREN],
					bw_nocken_zylinder_ausfahren := nockenschaltwerk_bestueckachse.fb.arr_spur[SP_BW_BANDKLEMMEN_BAWEV2_AUSFAHREN],
					uw_nocken_zylinder_einfahren :=  ,
					uw_nocken_zylinder_ausfahren :=  ,
					st_ctrl_out=> zyl_bandklemmen.st_ctrl.out,
					a_ventil_einfahren=> a_zyl_klemmen_einfahren,
					a_ventil_ausfahren=> );

				IF NOT gst_datensatz.st_md.b_auswahlSpruehoeler THEN
					zyl_oelen_oben.fb(
						st_config:= ,
						e_druckwaechter:= ST_Betriebsfreigaben.e_druckwaechter,
						i16_betriebsart:= gi16_betriebsart,
						b_no_gesteuert_im_norm_betrieb:= ,
						b_direkttaste_ausfahren:= ,
						b_direkttaste_mittefahren:= ,
						b_direkttaste_einfahren	:= ,
						st_ctrl_in:=zyl_oelen_oben.st_ctrl.in ,
						b_masterachse_hand_dialog_aktiv:=ST_Bestueckachse.b_hand_dialog_aktiv,
						st_visu:= visu.st_zyl,
						bw_nocken_zylinder_einfahren := (*ST_BandoelerZylinder.b_zyl_oben = FALSE OR*) nockenschaltwerk_bestueckachse.fb.arr_spur[56],
						bw_nocken_zylinder_ausfahren := (*ST_BandoelerZylinder.b_zyl_oben = TRUE AND*)  nockenschaltwerk_bestueckachse.fb.arr_spur[57],
						uw_nocken_zylinder_einfahren := zyl_oelen_oben.fb.e_sensor1_eingefahren AND  nockenschaltwerk_bestueckachse.fb.arr_spur[58],
						uw_nocken_zylinder_ausfahren := zyl_oelen_oben.fb.e_sensor1_ausgefahren AND  nockenschaltwerk_bestueckachse.fb.arr_spur[59],
						st_ctrl_out=> zyl_oelen_oben.st_ctrl.out,
						a_ventil_einfahren=> ,
						a_ventil_ausfahren=> );
	
					gst_datensatz.st_wkz.nockenschaltwerk_bestueckachse.arr_nocken[56].b_camvalid := TRUE;
					gst_datensatz.st_wkz.nockenschaltwerk_bestueckachse.arr_nocken[57].b_camvalid := TRUE;
					gst_datensatz.st_wkz.nockenschaltwerk_bestueckachse.arr_nocken[58].b_camvalid := TRUE;
					gst_datensatz.st_wkz.nockenschaltwerk_bestueckachse.arr_nocken[59].b_camvalid := TRUE;
	
					zyl_oelen_unten.fb(
						st_config:= ,
						e_druckwaechter:= ST_Betriebsfreigaben.e_druckwaechter,
						i16_betriebsart:= gi16_betriebsart,
						b_no_gesteuert_im_norm_betrieb:= ,
						b_direkttaste_ausfahren:= ,
						b_direkttaste_mittefahren:= ,
						b_direkttaste_einfahren	:= ,
						st_ctrl_in:=zyl_oelen_unten.st_ctrl.in ,
						b_masterachse_hand_dialog_aktiv:=ST_Bestueckachse.b_hand_dialog_aktiv,
						st_visu:= visu.st_zyl,
						bw_nocken_zylinder_einfahren := nockenschaltwerk_bestueckachse.fb.arr_spur[60],
						bw_nocken_zylinder_ausfahren := nockenschaltwerk_bestueckachse.fb.arr_spur[61],
						uw_nocken_zylinder_einfahren := zyl_oelen_unten.fb.e_sensor1_eingefahren AND nockenschaltwerk_bestueckachse.fb.arr_spur[62],
						uw_nocken_zylinder_ausfahren := zyl_oelen_unten.fb.e_sensor1_ausgefahren AND  nockenschaltwerk_bestueckachse.fb.arr_spur[63],
						st_ctrl_out=>zyl_oelen_unten.st_ctrl.out ,
						a_ventil_einfahren=> ,
						a_ventil_ausfahren=> );
	
					gst_datensatz.st_wkz.nockenschaltwerk_bestueckachse.arr_nocken[60].b_camvalid := TRUE;
					gst_datensatz.st_wkz.nockenschaltwerk_bestueckachse.arr_nocken[61].b_camvalid := TRUE;
					gst_datensatz.st_wkz.nockenschaltwerk_bestueckachse.arr_nocken[62].b_camvalid := TRUE;
					gst_datensatz.st_wkz.nockenschaltwerk_bestueckachse.arr_nocken[63].b_camvalid := TRUE;
				END_IF

			SERVO:
				;
		END_CASE

	BESTUECKZELLE_1720:
		ST_Datainit_Fast_Zylinder();

		CASE gst_datensatz.st_wkz.i16_typ_bandeinzug OF
			KEIN_EINZUG:
				;
		
			STANDARD_2FACH_V2:
				zyl_bandfaenger_li.fb(
					st_config:= ,
					e_druckwaechter:= ST_Betriebsfreigaben.e_druckwaechter,
					i16_betriebsart:= gi16_betriebsart,
					b_no_gesteuert_im_norm_betrieb:= ,
					b_direkttaste_ausfahren:= ,
					b_direkttaste_mittefahren:= ,
					b_direkttaste_einfahren	:= ,
					st_ctrl_in:= zyl_bandfaenger_li.st_ctrl.in,
					b_masterachse_hand_dialog_aktiv:= ST_Bestueckachse.b_hand_dialog_aktiv,
					st_visu:= visu.st_zyl,
					bw_nocken_zylinder_einfahren := nockenschaltwerk_bestueckachse.fb.arr_spur[SP_BW_BANDFAENGER_LI_BAEZV2_EINFAHREN],
					bw_nocken_zylinder_ausfahren := nockenschaltwerk_bestueckachse.fb.arr_spur[SP_BW_BANDFAENGER_LI_BAEZV2_AUSFAHREN],
					uw_nocken_zylinder_einfahren := ,
					uw_nocken_zylinder_ausfahren := ,
					st_ctrl_out=> zyl_bandfaenger_li.st_ctrl.out,
					a_ventil_einfahren=> ,
					a_ventil_ausfahren=> );
				
				zyl_bandfaenger_re.fb(
					st_config:= ,
					e_druckwaechter:= ST_Betriebsfreigaben.e_druckwaechter,
					i16_betriebsart:= gi16_betriebsart,
					b_no_gesteuert_im_norm_betrieb:= ,
					b_direkttaste_ausfahren:= ,
					b_direkttaste_mittefahren:= ,
					b_direkttaste_einfahren	:= ,
					st_ctrl_in:= zyl_bandfaenger_re.st_ctrl.in,
					b_masterachse_hand_dialog_aktiv:= ST_Bestueckachse.b_hand_dialog_aktiv,
					st_visu:= visu.st_zyl,
					bw_nocken_zylinder_einfahren := nockenschaltwerk_bestueckachse.fb.arr_spur[SP_BW_BANDFAENGER_RE_BAEZV2_EINFAHREN],
					bw_nocken_zylinder_ausfahren := nockenschaltwerk_bestueckachse.fb.arr_spur[SP_BW_BANDFAENGER_RE_BAEZV2_AUSFAHREN],
					uw_nocken_zylinder_einfahren := ,
					uw_nocken_zylinder_ausfahren := ,
					st_ctrl_out=> zyl_bandfaenger_re.st_ctrl.out,
					a_ventil_einfahren=> ,
					a_ventil_ausfahren=> );
		
				zyl_bandklemmen_li.fb(
					st_config:= ,
					e_druckwaechter:= ST_Betriebsfreigaben.e_druckwaechter,
					i16_betriebsart:= gi16_betriebsart,
					b_no_gesteuert_im_norm_betrieb:= ,
					b_direkttaste_ausfahren:= ,
					b_direkttaste_mittefahren:= ,
					b_direkttaste_einfahren	:= ,
					st_ctrl_in:= zyl_bandklemmen_li.st_ctrl.in,
					b_masterachse_hand_dialog_aktiv:= ST_Bestueckachse.b_hand_dialog_aktiv,
					st_visu:= visu.st_zyl,
					bw_nocken_zylinder_einfahren := nockenschaltwerk_bestueckachse.fb.arr_spur[SP_BW_BANDKLEMMEN_LI_BAEZV2_EINFAHREN],
					bw_nocken_zylinder_ausfahren := nockenschaltwerk_bestueckachse.fb.arr_spur[SP_BW_BANDKLEMMEN_LI_BAEZV2_AUSFAHREN],
					uw_nocken_zylinder_einfahren := ,
					uw_nocken_zylinder_ausfahren := ,
					st_ctrl_out=> zyl_bandklemmen_li.st_ctrl.out,
					a_ventil_einfahren=> ,
					a_ventil_ausfahren=> );
				
				zyl_bandklemmen_re.fb(
					st_config:= ,
					e_druckwaechter:= ST_Betriebsfreigaben.e_druckwaechter,
					i16_betriebsart:= gi16_betriebsart,
					b_no_gesteuert_im_norm_betrieb:= ,
					b_direkttaste_ausfahren:= ,
					b_direkttaste_mittefahren:= ,
					b_direkttaste_einfahren	:= ,
					st_ctrl_in:= zyl_bandklemmen_re.st_ctrl.in,
					b_masterachse_hand_dialog_aktiv:= ST_Bestueckachse.b_hand_dialog_aktiv,
					st_visu:= visu.st_zyl,
					bw_nocken_zylinder_einfahren := nockenschaltwerk_bestueckachse.fb.arr_spur[SP_BW_BANDKLEMMEN_RE_BAEZV2_EINFAHREN],
					bw_nocken_zylinder_ausfahren := nockenschaltwerk_bestueckachse.fb.arr_spur[SP_BW_BANDKLEMMEN_RE_BAEZV2_AUSFAHREN],
					uw_nocken_zylinder_einfahren := ,
					uw_nocken_zylinder_ausfahren := ,
					st_ctrl_out=> zyl_bandklemmen_re.st_ctrl.out,
					a_ventil_einfahren=> ,
					a_ventil_ausfahren=> );

			BANDWECHSLER_V2:
				;

			SERVO:
				;
		END_CASE;

	RASTERFOLIE:
		;
END_CASE
END_PROGRAM

(* POU Gemeinsamkeiten17xx/Initialisierung/Startup/ST_Datainit_Fast_Zylinder, ST *)
PROGRAM ST_Datainit_Fast_Zylinder
VAR
	b_config_fertig			: BOOL := FALSE;
END_VAR
CASE gst_datensatz.st_md.i16_typ_zelle OF
	KEINE_ZELLE:
 		;
	BESTUECKZELLE_1700:
		IF 	NOT zyl_bandfaenger.fb.st_config.b_config_fertig OR
			NOT zyl_bandklemmen.fb.st_config.b_config_fertig OR
			NOT zyl_oelen_unten.fb.st_config.b_config_fertig OR
			NOT zyl_oelen_oben.fb.st_config.b_config_fertig THEN


					(*Banölen unten*)
					zyl_oelen_unten.fb.st_config.b_config_fertig := FALSE;
					zyl_oelen_unten.fb.st_config.b_endlage1_aktiv := FALSE;
					zyl_oelen_unten.fb.st_config.b_endlage2_aktiv := FALSE;
					zyl_oelen_unten.fb.st_config.b_sensor1_aktiv := FALSE;
					zyl_oelen_unten.fb.st_config.b_sensor2_aktiv := FALSE;
					zyl_oelen_unten.fb.st_config.i16_gruppe := 1;
					zyl_oelen_unten.fb.st_config.i16_identnummer :=45;
					zyl_oelen_unten.fb.st_config.i16_meld_startindex := 2880;
					zyl_oelen_unten.fb.st_config.str_beschreibung := ' ';
					zyl_oelen_unten.fb.st_config.str_instanz_name := 'Bandoelen unten';
					zyl_oelen_unten.fb.st_config.str_zylinder_typ := '1V2E_EIN_AUS'; (*1V2E_EIN_AUS*)
					zyl_oelen_unten.fb.st_config.t_ein_aus_fahrzeit := t#100ms;
					zyl_oelen_unten.fb.st_config.t_ueberwachungszeit := t#1500ms;
					zyl_oelen_unten.fb.st_config.i16_tzk_faktor_ausfahren := 100;
					zyl_oelen_unten.fb.st_config.i16_tzk_faktor_einfahren := 100;
					zyl_oelen_unten.fb.st_config.b_config_fertig := TRUE;

					(*Banölen oben*)
					zyl_oelen_oben.fb.st_config.b_config_fertig := FALSE;
					zyl_oelen_oben.fb.st_config.b_endlage1_aktiv := FALSE;
					zyl_oelen_oben.fb.st_config.b_endlage2_aktiv := FALSE;
					zyl_oelen_oben.fb.st_config.b_sensor1_aktiv := FALSE;
					zyl_oelen_oben.fb.st_config.b_sensor2_aktiv := FALSE;
					zyl_oelen_oben.fb.st_config.i16_gruppe := 1;
					zyl_oelen_oben.fb.st_config.i16_identnummer :=46 ;
					zyl_oelen_oben.fb.st_config.i16_meld_startindex := 2900;
					zyl_oelen_oben.fb.st_config.str_beschreibung := ' ';
					zyl_oelen_oben.fb.st_config.str_instanz_name := 'Bandoelen oben';
					zyl_oelen_oben.fb.st_config.str_zylinder_typ := '1V2E_EIN_AUS'; (*1V2E_EIN_AUS*)
					zyl_oelen_oben.fb.st_config.t_ein_aus_fahrzeit := t#100ms;
					zyl_oelen_oben.fb.st_config.t_ueberwachungszeit := t#1500ms;
					zyl_oelen_oben.fb.st_config.i16_tzk_faktor_ausfahren := 100;
					zyl_oelen_oben.fb.st_config.i16_tzk_faktor_einfahren := 100;
					zyl_oelen_oben.fb.st_config.b_config_fertig := TRUE;

				(* Abhängig vom Bandwechseltyp *)
				CASE gst_datensatz.st_wkz.i16_typ_bandeinzug OF
					KEIN_EINZUG:
						;

					STANDARD_2FACH_V2:
						;

					BANDWECHSLER_V2:
						(* 1700: Bandfaenger *)
						zyl_bandfaenger.fb.st_config.b_config_fertig := FALSE;
						zyl_bandfaenger.fb.st_config.b_endlage1_aktiv := FALSE;
						zyl_bandfaenger.fb.st_config.b_endlage2_aktiv := FALSE;
						zyl_bandfaenger.fb.st_config.b_sensor1_aktiv := FALSE;
						zyl_bandfaenger.fb.st_config.b_sensor2_aktiv := FALSE;
						zyl_bandfaenger.fb.st_config.i16_gruppe := 1;
						zyl_bandfaenger.fb.st_config.i16_identnummer := 5;
						zyl_bandfaenger.fb.st_config.i16_meld_startindex := 2080;
						zyl_bandfaenger.fb.st_config.str_beschreibung := ' ';
						zyl_bandfaenger.fb.st_config.str_instanz_name := 'Bandfänger';
						zyl_bandfaenger.fb.st_config.str_zylinder_typ := '1V0E_NO';
						zyl_bandfaenger.fb.st_config.t_ein_aus_fahrzeit := t#0ms;
						zyl_bandfaenger.fb.st_config.t_ueberwachungszeit := t#500ms;
						zyl_bandfaenger.fb.st_config.i16_tzk_faktor_ausfahren := 100;
						zyl_bandfaenger.fb.st_config.i16_tzk_faktor_einfahren := 100;
						zyl_bandfaenger.fb.st_config.b_config_fertig := TRUE;
						(* 1700: Bandklemmen *)
						zyl_bandklemmen.fb.st_config.b_config_fertig := FALSE;
						zyl_bandklemmen.fb.st_config.b_endlage1_aktiv := FALSE;
						zyl_bandklemmen.fb.st_config.b_endlage2_aktiv := FALSE;
						zyl_bandklemmen.fb.st_config.b_sensor1_aktiv := FALSE;
						zyl_bandklemmen.fb.st_config.b_sensor2_aktiv := FALSE;
						zyl_bandklemmen.fb.st_config.i16_gruppe := 1;
						zyl_bandklemmen.fb.st_config.i16_identnummer := 6;
						zyl_bandklemmen.fb.st_config.i16_meld_startindex := 2100;
						zyl_bandklemmen.fb.st_config.str_beschreibung := ' ';
						zyl_bandklemmen.fb.st_config.str_instanz_name := 'Bandklemmen';
						zyl_bandklemmen.fb.st_config.str_zylinder_typ := '1V0E_NO';
						zyl_bandklemmen.fb.st_config.t_ein_aus_fahrzeit := t#0ms;
						zyl_bandklemmen.fb.st_config.t_ueberwachungszeit := t#500ms;
						zyl_bandklemmen.fb.st_config.i16_tzk_faktor_ausfahren := 100;
						zyl_bandklemmen.fb.st_config.i16_tzk_faktor_einfahren := 100;
						zyl_bandklemmen.fb.st_config.b_config_fertig := TRUE;

					SERVO:
						;
				END_CASE
		ELSE
			b_config_fertig := FALSE;
		END_IF

	BESTUECKZELLE_1720:
		IF 	NOT zyl_bandfaenger_li.fb.st_config.b_config_fertig OR
			NOT zyl_bandfaenger_re.fb.st_config.b_config_fertig OR
			NOT zyl_bandklemmen_li.fb.st_config.b_config_fertig OR
			NOT zyl_bandklemmen_re.fb.st_config.b_config_fertig
			THEN
				(* Abhängig vom Bandwechseltyp *)
				CASE gst_datensatz.st_wkz.i16_typ_bandeinzug OF
					KEIN_EINZUG:
						;

					STANDARD_2FACH_V2:
						(* 1720: Bandfaenger links *)
						zyl_bandfaenger_li.fb.st_config.b_config_fertig := FALSE;
						zyl_bandfaenger_li.fb.st_config.b_endlage1_aktiv := FALSE;
						zyl_bandfaenger_li.fb.st_config.b_endlage2_aktiv := FALSE;
						zyl_bandfaenger_li.fb.st_config.b_sensor1_aktiv := FALSE;
						zyl_bandfaenger_li.fb.st_config.b_sensor2_aktiv := FALSE;
						zyl_bandfaenger_li.fb.st_config.i16_gruppe := 1;
						zyl_bandfaenger_li.fb.st_config.i16_identnummer := 1;
						zyl_bandfaenger_li.fb.st_config.i16_meld_startindex := 2000;
						zyl_bandfaenger_li.fb.st_config.str_beschreibung := ' ';
						zyl_bandfaenger_li.fb.st_config.str_instanz_name := 'Bandfänger links';
						zyl_bandfaenger_li.fb.st_config.str_zylinder_typ := '1V0E_NO';
						zyl_bandfaenger_li.fb.st_config.t_ein_aus_fahrzeit := t#0ms;
						zyl_bandfaenger_li.fb.st_config.t_ueberwachungszeit := t#500ms;
						zyl_bandfaenger_li.fb.st_config.i16_tzk_faktor_ausfahren := 100;
						zyl_bandfaenger_li.fb.st_config.i16_tzk_faktor_einfahren := 100;
						zyl_bandfaenger_li.fb.st_config.b_config_fertig := TRUE;
						(* 1720: Bandfaenger rechts *)
						zyl_bandfaenger_re.fb.st_config.b_config_fertig := FALSE;
						zyl_bandfaenger_re.fb.st_config.b_endlage1_aktiv := FALSE;
						zyl_bandfaenger_re.fb.st_config.b_endlage2_aktiv := FALSE;
						zyl_bandfaenger_re.fb.st_config.b_sensor1_aktiv := FALSE;
						zyl_bandfaenger_re.fb.st_config.b_sensor2_aktiv := FALSE;
						zyl_bandfaenger_re.fb.st_config.i16_gruppe := 1;
						zyl_bandfaenger_re.fb.st_config.i16_identnummer := 2;
						zyl_bandfaenger_re.fb.st_config.i16_meld_startindex := 2020;
						zyl_bandfaenger_re.fb.st_config.str_beschreibung := ' ';
						zyl_bandfaenger_re.fb.st_config.str_instanz_name := 'Bandfänger rechts';
						zyl_bandfaenger_re.fb.st_config.str_zylinder_typ := '1V0E_NO';
						zyl_bandfaenger_re.fb.st_config.t_ein_aus_fahrzeit := t#0ms;
						zyl_bandfaenger_re.fb.st_config.t_ueberwachungszeit := t#500ms;
						zyl_bandfaenger_re.fb.st_config.i16_tzk_faktor_ausfahren := 100;
						zyl_bandfaenger_re.fb.st_config.i16_tzk_faktor_einfahren := 100;
						zyl_bandfaenger_re.fb.st_config.b_config_fertig := TRUE;
						
